//     PlcTask Outputs/G_IO.arDO[20]/Ch[11] <-> DO0/0016ETP Output-bit maping/Digital output CH2-bit3
//     PlcTask Outputs/G_IO.arDO[20]/Ch[12] <-> DO0/0016ETP Output-bit maping/Digital output CH2-bit4
//     PlcTask Outputs/G_IO.arDO[20]/Ch[13] <-> DO0/0016ETP Output-bit maping/Digital output CH2-bit5
//     PlcTask Outputs/G_IO.arDO[20]/Ch[14] <-> DO0/0016ETP Output-bit maping/Digital output CH2-bit6
//     PlcTask Outputs/G_IO.arDO[20]/Ch[15] <-> DO0/0016ETP Output-bit maping/Digital output CH2-bit7
//     PlcTask Outputs/G_IO.arDO[20]/Ch[1] <-> DO0/0016ETP Output-bit maping/Digital output CH1-bit1
//     PlcTask Outputs/G_IO.arDO[20]/Ch[2] <-> DO0/0016ETP Output-bit maping/Digital output CH1-bit2
//     PlcTask Outputs/G_IO.arDO[20]/Ch[3] <-> DO0/0016ETP Output-bit maping/Digital output CH1-bit3
//     PlcTask Outputs/G_IO.arDO[20]/Ch[4] <-> DO0/0016ETP Output-bit maping/Digital output CH1-bit4
//     PlcTask Outputs/G_IO.arDO[20]/Ch[5] <-> DO0/0016ETP Output-bit maping/Digital output CH1-bit5
//     PlcTask Outputs/G_IO.arDO[20]/Ch[6] <-> DO0/0016ETP Output-bit maping/Digital output CH1-bit6
//     PlcTask Outputs/G_IO.arDO[20]/Ch[7] <-> DO0/0016ETP Output-bit maping/Digital output CH1-bit7
//     PlcTask Outputs/G_IO.arDO[20]/Ch[8] <-> DO0/0016ETP Output-bit maping/Digital output CH2-bit0
//     PlcTask Outputs/G_IO.arDO[20]/Ch[9] <-> DO0/0016ETP Output-bit maping/Digital output CH2-bit1
//     PlcTask Outputs/G_IO.arDO[21]/Ch[0] <-> DO1/0016ETP Output-bit maping/Digital output CH1-bit0
//     PlcTask Outputs/G_IO.arDO[21]/Ch[10] <-> DO1/0016ETP Output-bit maping/Digital output CH2-bit2
//     PlcTask Outputs/G_IO.arDO[21]/Ch[11] <-> DO1/0016ETP Output-bit maping/Digital output CH2-bit3
//     PlcTask Outputs/G_IO.arDO[21]/Ch[12] <-> DO1/0016ETP Output-bit maping/Digital output CH2-bit4
//     PlcTask Outputs/G_IO.arDO[21]/Ch[13] <-> DO1/0016ETP Output-bit maping/Digital output CH2-bit5
//     PlcTask Outputs/G_IO.arDO[21]/Ch[14] <-> DO1/0016ETP Output-bit maping/Digital output CH2-bit6
//     PlcTask Outputs/G_IO.arDO[21]/Ch[15] <-> DO1/0016ETP Output-bit maping/Digital output CH2-bit7
//     PlcTask Outputs/G_IO.arDO[21]/Ch[1] <-> DO1/0016ETP Output-bit maping/Digital output CH1-bit1
//     PlcTask Outputs/G_IO.arDO[21]/Ch[2] <-> DO1/0016ETP Output-bit maping/Digital output CH1-bit2
//     PlcTask Outputs/G_IO.arDO[21]/Ch[3] <-> DO1/0016ETP Output-bit maping/Digital output CH1-bit3
//     PlcTask Outputs/G_IO.arDO[21]/Ch[4] <-> DO1/0016ETP Output-bit maping/Digital output CH1-bit4
//     PlcTask Outputs/G_IO.arDO[21]/Ch[5] <-> DO1/0016ETP Output-bit maping/Digital output CH1-bit5
//     PlcTask Outputs/G_IO.arDO[21]/Ch[6] <-> DO1/0016ETP Output-bit maping/Digital output CH1-bit6
//     PlcTask Outputs/G_IO.arDO[21]/Ch[7] <-> DO1/0016ETP Output-bit maping/Digital output CH1-bit7
//     PlcTask Outputs/G_IO.arDO[21]/Ch[8] <-> DO1/0016ETP Output-bit maping/Digital output CH2-bit0
//     PlcTask Outputs/G_IO.arDO[21]/Ch[9] <-> DO1/0016ETP Output-bit maping/Digital output CH2-bit1
//   kittingDeca/kittingDeca Instance <-> rem_wf/rem5_valve
//     PlcTask Outputs/G_IO.arDO[22]/Ch[0] <-> Module 1 (C2S-EC-24B)/Outputs/valve[1..4][0]
//     PlcTask Outputs/G_IO.arDO[22]/Ch[10] <-> Module 1 (C2S-EC-24B)/Outputs/valve[5..8][2]
//     PlcTask Outputs/G_IO.arDO[22]/Ch[11] <-> Module 1 (C2S-EC-24B)/Outputs/valve[5..8][3]
//     PlcTask Outputs/G_IO.arDO[22]/Ch[12] <-> Module 1 (C2S-EC-24B)/Outputs/valve[5..8][4]
//     PlcTask Outputs/G_IO.arDO[22]/Ch[13] <-> Module 1 (C2S-EC-24B)/Outputs/valve[5..8][5]
//     PlcTask Outputs/G_IO.arDO[22]/Ch[14] <-> Module 1 (C2S-EC-24B)/Outputs/valve[5..8][6]
//     PlcTask Outputs/G_IO.arDO[22]/Ch[15] <-> Module 1 (C2S-EC-24B)/Outputs/valve[5..8][7]
//     PlcTask Outputs/G_IO.arDO[22]/Ch[1] <-> Module 1 (C2S-EC-24B)/Outputs/valve[1..4][1]
//     PlcTask Outputs/G_IO.arDO[22]/Ch[2] <-> Module 1 (C2S-EC-24B)/Outputs/valve[1..4][2]
//     PlcTask Outputs/G_IO.arDO[22]/Ch[3] <-> Module 1 (C2S-EC-24B)/Outputs/valve[1..4][3]
//     PlcTask Outputs/G_IO.arDO[22]/Ch[4] <-> Module 1 (C2S-EC-24B)/Outputs/valve[1..4][4]
//     PlcTask Outputs/G_IO.arDO[22]/Ch[5] <-> Module 1 (C2S-EC-24B)/Outputs/valve[1..4][5]
//     PlcTask Outputs/G_IO.arDO[22]/Ch[6] <-> Module 1 (C2S-EC-24B)/Outputs/valve[1..4][6]
//     PlcTask Outputs/G_IO.arDO[22]/Ch[7] <-> Module 1 (C2S-EC-24B)/Outputs/valve[1..4][7]
//     PlcTask Outputs/G_IO.arDO[22]/Ch[8] <-> Module 1 (C2S-EC-24B)/Outputs/valve[5..8][0]
//     PlcTask Outputs/G_IO.arDO[22]/Ch[9] <-> Module 1 (C2S-EC-24B)/Outputs/valve[5..8][1]
//     PlcTask Outputs/G_IO.arDO[23]/Ch[0] <-> Module 1 (C2S-EC-24B)/Outputs/valve[9..12][0]
//     PlcTask Outputs/G_IO.arDO[23]/Ch[1] <-> Module 1 (C2S-EC-24B)/Outputs/valve[9..12][1]
//     PlcTask Outputs/G_IO.arDO[23]/Ch[2] <-> Module 1 (C2S-EC-24B)/Outputs/valve[9..12][2]
//     PlcTask Outputs/G_IO.arDO[23]/Ch[3] <-> Module 1 (C2S-EC-24B)/Outputs/valve[9..12][3]
//     PlcTask Outputs/G_IO.arDO[23]/Ch[4] <-> Module 1 (C2S-EC-24B)/Outputs/valve[9..12][4]
//     PlcTask Outputs/G_IO.arDO[23]/Ch[5] <-> Module 1 (C2S-EC-24B)/Outputs/valve[9..12][5]
//     PlcTask Outputs/G_IO.arDO[23]/Ch[6] <-> Module 1 (C2S-EC-24B)/Outputs/valve[9..12][6]
//     PlcTask Outputs/G_IO.arDO[23]/Ch[7] <-> Module 1 (C2S-EC-24B)/Outputs/valve[9..12][7]
//   kittingDeca/kittingDeca Instance <-> rem_wf/rem6_dio
//     PlcTask Inputs/G_IO.arDI[24]/Ch[0] <-> DI0/1600END input-bit maping/Digital input CH1-bit0
//     PlcTask Inputs/G_IO.arDI[24]/Ch[10] <-> DI0/1600END input-bit maping/Digital input CH2-bit2
//     PlcTask Inputs/G_IO.arDI[24]/Ch[11] <-> DI0/1600END input-bit maping/Digital input CH2-bit3
//     PlcTask Inputs/G_IO.arDI[24]/Ch[12] <-> DI0/1600END input-bit maping/Digital input CH2-bit4
//     PlcTask Inputs/G_IO.arDI[24]/Ch[13] <-> DI0/1600END input-bit maping/Digital input CH2-bit5
//     PlcTask Inputs/G_IO.arDI[24]/Ch[14] <-> DI0/1600END input-bit maping/Digital input CH2-bit6
//     PlcTask Inputs/G_IO.arDI[24]/Ch[15] <-> DI0/1600END input-bit maping/Digital input CH2-bit7
//     PlcTask Inputs/G_IO.arDI[24]/Ch[1] <-> DI0/1600END input-bit maping/Digital input CH1-bit1
//     PlcTask Inputs/G_IO.arDI[24]/Ch[2] <-> DI0/1600END input-bit maping/Digital input CH1-bit2
//     PlcTask Inputs/G_IO.arDI[24]/Ch[3] <-> DI0/1600END input-bit maping/Digital input CH1-bit3
//     PlcTask Inputs/G_IO.arDI[24]/Ch[4] <-> DI0/1600END input-bit maping/Digital input CH1-bit4
//     PlcTask Inputs/G_IO.arDI[24]/Ch[5] <-> DI0/1600END input-bit maping/Digital input CH1-bit5
//     PlcTask Inputs/G_IO.arDI[24]/Ch[6] <-> DI0/1600END input-bit maping/Digital input CH1-bit6
//     PlcTask Inputs/G_IO.arDI[24]/Ch[7] <-> DI0/1600END input-bit maping/Digital input CH1-bit7
//     PlcTask Inputs/G_IO.arDI[24]/Ch[8] <-> DI0/1600END input-bit maping/Digital input CH2-bit0
//     PlcTask Inputs/G_IO.arDI[24]/Ch[9] <-> DI0/1600END input-bit maping/Digital input CH2-bit1
//     PlcTask Inputs/G_IO.arDI[25]/Ch[0] <-> DI1/1600END input-bit maping/Digital input CH1-bit0
//     PlcTask Inputs/G_IO.arDI[25]/Ch[10] <-> DI1/1600END input-bit maping/Digital input CH2-bit2
//     PlcTask Inputs/G_IO.arDI[25]/Ch[11] <-> DI1/1600END input-bit maping/Digital input CH2-bit3
//     PlcTask Inputs/G_IO.arDI[25]/Ch[12] <-> DI1/1600END input-bit maping/Digital input CH2-bit4
//     PlcTask Inputs/G_IO.arDI[25]/Ch[13] <-> DI1/1600END input-bit maping/Digital input CH2-bit5
//     PlcTask Inputs/G_IO.arDI[25]/Ch[14] <-> DI1/1600END input-bit maping/Digital input CH2-bit6
//     PlcTask Inputs/G_IO.arDI[25]/Ch[15] <-> DI1/1600END input-bit maping/Digital input CH2-bit7
//     PlcTask Inputs/G_IO.arDI[25]/Ch[1] <-> DI1/1600END input-bit maping/Digital input CH1-bit1
//     PlcTask Inputs/G_IO.arDI[25]/Ch[2] <-> DI1/1600END input-bit maping/Digital input CH1-bit2
//     PlcTask Inputs/G_IO.arDI[25]/Ch[3] <-> DI1/1600END input-bit maping/Digital input CH1-bit3
//     PlcTask Inputs/G_IO.arDI[25]/Ch[4] <-> DI1/1600END input-bit maping/Digital input CH1-bit4
//     PlcTask Inputs/G_IO.arDI[25]/Ch[5] <-> DI1/1600END input-bit maping/Digital input CH1-bit5
//     PlcTask Inputs/G_IO.arDI[25]/Ch[6] <-> DI1/1600END input-bit maping/Digital input CH1-bit6
//     PlcTask Inputs/G_IO.arDI[25]/Ch[7] <-> DI1/1600END input-bit maping/Digital input CH1-bit7
//     PlcTask Inputs/G_IO.arDI[25]/Ch[8] <-> DI1/1600END input-bit maping/Digital input CH2-bit0
//     PlcTask Inputs/G_IO.arDI[25]/Ch[9] <-> DI1/1600END input-bit maping/Digital input CH2-bit1
//     PlcTask Inputs/G_IO.arDI[26]/Ch[0] <-> DI2/1600END input-bit maping/Digital input CH1-bit0
//     PlcTask Inputs/G_IO.arDI[26]/Ch[10] <-> DI2/1600END input-bit maping/Digital input CH2-bit2
//     PlcTask Inputs/G_IO.arDI[26]/Ch[11] <-> DI2/1600END input-bit maping/Digital input CH2-bit3
//     PlcTask Inputs/G_IO.arDI[26]/Ch[12] <-> DI2/1600END input-bit maping/Digital input CH2-bit4
//     PlcTask Inputs/G_IO.arDI[26]/Ch[13] <-> DI2/1600END input-bit maping/Digital input CH2-bit5
//     PlcTask Inputs/G_IO.arDI[26]/Ch[14] <-> DI2/1600END input-bit maping/Digital input CH2-bit6
//     PlcTask Inputs/G_IO.arDI[26]/Ch[15] <-> DI2/1600END input-bit maping/Digital input CH2-bit7
//     PlcTask Inputs/G_IO.arDI[26]/Ch[1] <-> DI2/1600END input-bit maping/Digital input CH1-bit1
//     PlcTask Inputs/G_IO.arDI[26]/Ch[2] <-> DI2/1600END input-bit maping/Digital input CH1-bit2
//     PlcTask Inputs/G_IO.arDI[26]/Ch[3] <-> DI2/1600END input-bit maping/Digital input CH1-bit3
//     PlcTask Inputs/G_IO.arDI[26]/Ch[4] <-> DI2/1600END input-bit maping/Digital input CH1-bit4
//     PlcTask Inputs/G_IO.arDI[26]/Ch[5] <-> DI2/1600END input-bit maping/Digital input CH1-bit5
//     PlcTask Inputs/G_IO.arDI[26]/Ch[6] <-> DI2/1600END input-bit maping/Digital input CH1-bit6
//     PlcTask Inputs/G_IO.arDI[26]/Ch[7] <-> DI2/1600END input-bit maping/Digital input CH1-bit7
//     PlcTask Inputs/G_IO.arDI[26]/Ch[8] <-> DI2/1600END input-bit maping/Digital input CH2-bit0
//     PlcTask Inputs/G_IO.arDI[26]/Ch[9] <-> DI2/1600END input-bit maping/Digital input CH2-bit1
//     PlcTask Inputs/G_IO.arDI[27]/Ch[0] <-> DI3/1600END input-bit maping/Digital input CH1-bit0
//     PlcTask Inputs/G_IO.arDI[27]/Ch[10] <-> DI3/1600END input-bit maping/Digital input CH2-bit2
//     PlcTask Inputs/G_IO.arDI[27]/Ch[11] <-> DI3/1600END input-bit maping/Digital input CH2-bit3
//     PlcTask Inputs/G_IO.arDI[27]/Ch[12] <-> DI3/1600END input-bit maping/Digital input CH2-bit4
//     PlcTask Inputs/G_IO.arDI[27]/Ch[13] <-> DI3/1600END input-bit maping/Digital input CH2-bit5
//     PlcTask Inputs/G_IO.arDI[27]/Ch[14] <-> DI3/1600END input-bit maping/Digital input CH2-bit6
//     PlcTask Inputs/G_IO.arDI[27]/Ch[15] <-> DI3/1600END input-bit maping/Digital input CH2-bit7
//     PlcTask Inputs/G_IO.arDI[27]/Ch[1] <-> DI3/1600END input-bit maping/Digital input CH1-bit1
//     PlcTask Inputs/G_IO.arDI[27]/Ch[2] <-> DI3/1600END input-bit maping/Digital input CH1-bit2
//     PlcTask Inputs/G_IO.arDI[27]/Ch[3] <-> DI3/1600END input-bit maping/Digital input CH1-bit3
//     PlcTask Inputs/G_IO.arDI[27]/Ch[4] <-> DI3/1600END input-bit maping/Digital input CH1-bit4
//     PlcTask Inputs/G_IO.arDI[27]/Ch[5] <-> DI3/1600END input-bit maping/Digital input CH1-bit5
//     PlcTask Inputs/G_IO.arDI[27]/Ch[6] <-> DI3/1600END input-bit maping/Digital input CH1-bit6
//     PlcTask Inputs/G_IO.arDI[27]/Ch[7] <-> DI3/1600END input-bit maping/Digital input CH1-bit7
//     PlcTask Inputs/G_IO.arDI[27]/Ch[8] <-> DI3/1600END input-bit maping/Digital input CH2-bit0
//     PlcTask Inputs/G_IO.arDI[27]/Ch[9] <-> DI3/1600END input-bit maping/Digital input CH2-bit1
//     PlcTask Outputs/G_IO.arDO[24]/Ch[0] <-> DO0/0016ETP Output-bit maping/Digital output CH1-bit0
//     PlcTask Outputs/G_IO.arDO[24]/Ch[10] <-> DO0/0016ETP Output-bit maping/Digital output CH2-bit2
//     PlcTask Outputs/G_IO.arDO[24]/Ch[11] <-> DO0/0016ETP Output-bit maping/Digital output CH2-bit3
//     PlcTask Outputs/G_IO.arDO[24]/Ch[12] <-> DO0/0016ETP Output-bit maping/Digital output CH2-bit4
//     PlcTask Outputs/G_IO.arDO[24]/Ch[13] <-> DO0/0016ETP Output-bit maping/Digital output CH2-bit5
//     PlcTask Outputs/G_IO.arDO[24]/Ch[14] <-> DO0/0016ETP Output-bit maping/Digital output CH2-bit6
//     PlcTask Outputs/G_IO.arDO[24]/Ch[15] <-> DO0/0016ETP Output-bit maping/Digital output CH2-bit7
//     PlcTask Outputs/G_IO.arDO[24]/Ch[1] <-> DO0/0016ETP Output-bit maping/Digital output CH1-bit1
//     PlcTask Outputs/G_IO.arDO[24]/Ch[2] <-> DO0/0016ETP Output-bit maping/Digital output CH1-bit2
//     PlcTask Outputs/G_IO.arDO[24]/Ch[3] <-> DO0/0016ETP Output-bit maping/Digital output CH1-bit3
//     PlcTask Outputs/G_IO.arDO[24]/Ch[4] <-> DO0/0016ETP Output-bit maping/Digital output CH1-bit4
//     PlcTask Outputs/G_IO.arDO[24]/Ch[5] <-> DO0/0016ETP Output-bit maping/Digital output CH1-bit5
//     PlcTask Outputs/G_IO.arDO[24]/Ch[6] <-> DO0/0016ETP Output-bit maping/Digital output CH1-bit6
//     PlcTask Outputs/G_IO.arDO[24]/Ch[7] <-> DO0/0016ETP Output-bit maping/Digital output CH1-bit7
//     PlcTask Outputs/G_IO.arDO[24]/Ch[8] <-> DO0/0016ETP Output-bit maping/Digital output CH2-bit0
//     PlcTask Outputs/G_IO.arDO[24]/Ch[9] <-> DO0/0016ETP Output-bit maping/Digital output CH2-bit1
//     PlcTask Outputs/G_IO.arDO[25]/Ch[0] <-> DO1/0016ETP Output-bit maping/Digital output CH1-bit0
//     PlcTask Outputs/G_IO.arDO[25]/Ch[10] <-> DO1/0016ETP Output-bit maping/Digital output CH2-bit2
//     PlcTask Outputs/G_IO.arDO[25]/Ch[11] <-> DO1/0016ETP Output-bit maping/Digital output CH2-bit3
//     PlcTask Outputs/G_IO.arDO[25]/Ch[12] <-> DO1/0016ETP Output-bit maping/Digital output CH2-bit4
//     PlcTask Outputs/G_IO.arDO[25]/Ch[13] <-> DO1/0016ETP Output-bit maping/Digital output CH2-bit5
//     PlcTask Outputs/G_IO.arDO[25]/Ch[14] <-> DO1/0016ETP Output-bit maping/Digital output CH2-bit6
//     PlcTask Outputs/G_IO.arDO[25]/Ch[15] <-> DO1/0016ETP Output-bit maping/Digital output CH2-bit7
//     PlcTask Outputs/G_IO.arDO[25]/Ch[1] <-> DO1/0016ETP Output-bit maping/Digital output CH1-bit1
//     PlcTask Outputs/G_IO.arDO[25]/Ch[2] <-> DO1/0016ETP Output-bit maping/Digital output CH1-bit2
//     PlcTask Outputs/G_IO.arDO[25]/Ch[3] <-> DO1/0016ETP Output-bit maping/Digital output CH1-bit3
//     PlcTask Outputs/G_IO.arDO[25]/Ch[4] <-> DO1/0016ETP Output-bit maping/Digital output CH1-bit4
//     PlcTask Outputs/G_IO.arDO[25]/Ch[5] <-> DO1/0016ETP Output-bit maping/Digital output CH1-bit5
//     PlcTask Outputs/G_IO.arDO[25]/Ch[6] <-> DO1/0016ETP Output-bit maping/Digital output CH1-bit6
//     PlcTask Outputs/G_IO.arDO[25]/Ch[7] <-> DO1/0016ETP Output-bit maping/Digital output CH1-bit7
//     PlcTask Outputs/G_IO.arDO[25]/Ch[8] <-> DO1/0016ETP Output-bit maping/Digital output CH2-bit0
//     PlcTask Outputs/G_IO.arDO[25]/Ch[9] <-> DO1/0016ETP Output-bit maping/Digital output CH2-bit1
//   kittingDeca/kittingDeca Instance <-> rem_wf/rem6_valve
//     PlcTask Outputs/G_IO.arDO[26]/Ch[0] <-> Module 1 (C2S-EC-24B)/Outputs/valve[1..4][0]
//     PlcTask Outputs/G_IO.arDO[26]/Ch[10] <-> Module 1 (C2S-EC-24B)/Outputs/valve[5..8][2]
//     PlcTask Outputs/G_IO.arDO[26]/Ch[11] <-> Module 1 (C2S-EC-24B)/Outputs/valve[5..8][3]
//     PlcTask Outputs/G_IO.arDO[26]/Ch[12] <-> Module 1 (C2S-EC-24B)/Outputs/valve[5..8][4]
//     PlcTask Outputs/G_IO.arDO[26]/Ch[13] <-> Module 1 (C2S-EC-24B)/Outputs/valve[5..8][5]
//     PlcTask Outputs/G_IO.arDO[26]/Ch[14] <-> Module 1 (C2S-EC-24B)/Outputs/valve[5..8][6]
//     PlcTask Outputs/G_IO.arDO[26]/Ch[15] <-> Module 1 (C2S-EC-24B)/Outputs/valve[5..8][7]
//     PlcTask Outputs/G_IO.arDO[26]/Ch[1] <-> Module 1 (C2S-EC-24B)/Outputs/valve[1..4][1]
//     PlcTask Outputs/G_IO.arDO[26]/Ch[2] <-> Module 1 (C2S-EC-24B)/Outputs/valve[1..4][2]
//     PlcTask Outputs/G_IO.arDO[26]/Ch[3] <-> Module 1 (C2S-EC-24B)/Outputs/valve[1..4][3]
//     PlcTask Outputs/G_IO.arDO[26]/Ch[4] <-> Module 1 (C2S-EC-24B)/Outputs/valve[1..4][4]
//     PlcTask Outputs/G_IO.arDO[26]/Ch[5] <-> Module 1 (C2S-EC-24B)/Outputs/valve[1..4][5]
//     PlcTask Outputs/G_IO.arDO[26]/Ch[6] <-> Module 1 (C2S-EC-24B)/Outputs/valve[1..4][6]
//     PlcTask Outputs/G_IO.arDO[26]/Ch[7] <-> Module 1 (C2S-EC-24B)/Outputs/valve[1..4][7]
//     PlcTask Outputs/G_IO.arDO[26]/Ch[8] <-> Module 1 (C2S-EC-24B)/Outputs/valve[5..8][0]
//     PlcTask Outputs/G_IO.arDO[26]/Ch[9] <-> Module 1 (C2S-EC-24B)/Outputs/valve[5..8][1]
//     PlcTask Outputs/G_IO.arDO[27]/Ch[0] <-> Module 1 (C2S-EC-24B)/Outputs/valve[9..12][0]
//     PlcTask Outputs/G_IO.arDO[27]/Ch[1] <-> Module 1 (C2S-EC-24B)/Outputs/valve[9..12][1]
//     PlcTask Outputs/G_IO.arDO[27]/Ch[2] <-> Module 1 (C2S-EC-24B)/Outputs/valve[9..12][2]
//     PlcTask Outputs/G_IO.arDO[27]/Ch[3] <-> Module 1 (C2S-EC-24B)/Outputs/valve[9..12][3]
//     PlcTask Outputs/G_IO.arDO[27]/Ch[4] <-> Module 1 (C2S-EC-24B)/Outputs/valve[9..12][4]
//     PlcTask Outputs/G_IO.arDO[27]/Ch[5] <-> Module 1 (C2S-EC-24B)/Outputs/valve[9..12][5]
//     PlcTask Outputs/G_IO.arDO[27]/Ch[6] <-> Module 1 (C2S-EC-24B)/Outputs/valve[9..12][6]
//     PlcTask Outputs/G_IO.arDO[27]/Ch[7] <-> Module 1 (C2S-EC-24B)/Outputs/valve[9..12][7]
//   kittingDeca/kittingDeca Instance <-> rem_wf/rem7_dio
//     PlcTask Inputs/G_IO.arDI[28]/Ch[0] <-> DI0/1600END input-bit maping/Digital input CH1-bit0
//     PlcTask Inputs/G_IO.arDI[28]/Ch[10] <-> DI0/1600END input-bit maping/Digital input CH2-bit2
//     PlcTask Inputs/G_IO.arDI[28]/Ch[11] <-> DI0/1600END input-bit maping/Digital input CH2-bit3
//     PlcTask Inputs/G_IO.arDI[28]/Ch[12] <-> DI0/1600END input-bit maping/Digital input CH2-bit4
//     PlcTask Inputs/G_IO.arDI[28]/Ch[13] <-> DI0/1600END input-bit maping/Digital input CH2-bit5
//     PlcTask Inputs/G_IO.arDI[28]/Ch[14] <-> DI0/1600END input-bit maping/Digital input CH2-bit6
//     PlcTask Inputs/G_IO.arDI[28]/Ch[15] <-> DI0/1600END input-bit maping/Digital input CH2-bit7
//     PlcTask Inputs/G_IO.arDI[28]/Ch[1] <-> DI0/1600END input-bit maping/Digital input CH1-bit1
//     PlcTask Inputs/G_IO.arDI[28]/Ch[2] <-> DI0/1600END input-bit maping/Digital input CH1-bit2
//     PlcTask Inputs/G_IO.arDI[28]/Ch[3] <-> DI0/1600END input-bit maping/Digital input CH1-bit3
//     PlcTask Inputs/G_IO.arDI[28]/Ch[4] <-> DI0/1600END input-bit maping/Digital input CH1-bit4
//     PlcTask Inputs/G_IO.arDI[28]/Ch[5] <-> DI0/1600END input-bit maping/Digital input CH1-bit5
//     PlcTask Inputs/G_IO.arDI[28]/Ch[6] <-> DI0/1600END input-bit maping/Digital input CH1-bit6
//     PlcTask Inputs/G_IO.arDI[28]/Ch[7] <-> DI0/1600END input-bit maping/Digital input CH1-bit7
//     PlcTask Inputs/G_IO.arDI[28]/Ch[8] <-> DI0/1600END input-bit maping/Digital input CH2-bit0
//     PlcTask Inputs/G_IO.arDI[28]/Ch[9] <-> DI0/1600END input-bit maping/Digital input CH2-bit1
//     PlcTask Inputs/G_IO.arDI[29]/Ch[0] <-> DI1/1600END input-bit maping/Digital input CH1-bit0
//     PlcTask Inputs/G_IO.arDI[29]/Ch[10] <-> DI1/1600END input-bit maping/Digital input CH2-bit2
//     PlcTask Inputs/G_IO.arDI[29]/Ch[11] <-> DI1/1600END input-bit maping/Digital input CH2-bit3
//     PlcTask Inputs/G_IO.arDI[29]/Ch[12] <-> DI1/1600END input-bit maping/Digital input CH2-bit4
//     PlcTask Inputs/G_IO.arDI[29]/Ch[13] <-> DI1/1600END input-bit maping/Digital input CH2-bit5
//     PlcTask Inputs/G_IO.arDI[29]/Ch[14] <-> DI1/1600END input-bit maping/Digital input CH2-bit6
//     PlcTask Inputs/G_IO.arDI[29]/Ch[15] <-> DI1/1600END input-bit maping/Digital input CH2-bit7
//     PlcTask Inputs/G_IO.arDI[29]/Ch[1] <-> DI1/1600END input-bit maping/Digital input CH1-bit1
//     PlcTask Inputs/G_IO.arDI[29]/Ch[2] <-> DI1/1600END input-bit maping/Digital input CH1-bit2
//     PlcTask Inputs/G_IO.arDI[29]/Ch[3] <-> DI1/1600END input-bit maping/Digital input CH1-bit3
//     PlcTask Inputs/G_IO.arDI[29]/Ch[4] <-> DI1/1600END input-bit maping/Digital input CH1-bit4
//     PlcTask Inputs/G_IO.arDI[29]/Ch[5] <-> DI1/1600END input-bit maping/Digital input CH1-bit5
//     PlcTask Inputs/G_IO.arDI[29]/Ch[6] <-> DI1/1600END input-bit maping/Digital input CH1-bit6
//     PlcTask Inputs/G_IO.arDI[29]/Ch[7] <-> DI1/1600END input-bit maping/Digital input CH1-bit7
//     PlcTask Inputs/G_IO.arDI[29]/Ch[8] <-> DI1/1600END input-bit maping/Digital input CH2-bit0
//     PlcTask Inputs/G_IO.arDI[29]/Ch[9] <-> DI1/1600END input-bit maping/Digital input CH2-bit1
//     PlcTask Inputs/G_IO.arDI[30]/Ch[0] <-> DI2/1600END input-bit maping/Digital input CH1-bit0
//     PlcTask Inputs/G_IO.arDI[30]/Ch[10] <-> DI2/1600END input-bit maping/Digital input CH2-bit2
//     PlcTask Inputs/G_IO.arDI[30]/Ch[11] <-> DI2/1600END input-bit maping/Digital input CH2-bit3
//     PlcTask Inputs/G_IO.arDI[30]/Ch[12] <-> DI2/1600END input-bit maping/Digital input CH2-bit4
//     PlcTask Inputs/G_IO.arDI[30]/Ch[13] <-> DI2/1600END input-bit maping/Digital input CH2-bit5
//     PlcTask Inputs/G_IO.arDI[30]/Ch[14] <-> DI2/1600END input-bit maping/Digital input CH2-bit6
//     PlcTask Inputs/G_IO.arDI[30]/Ch[15] <-> DI2/1600END input-bit maping/Digital input CH2-bit7
//     PlcTask Inputs/G_IO.arDI[30]/Ch[1] <-> DI2/1600END input-bit maping/Digital input CH1-bit1
//     PlcTask Inputs/G_IO.arDI[30]/Ch[2] <-> DI2/1600END input-bit maping/Digital input CH1-bit2
//     PlcTask Inputs/G_IO.arDI[30]/Ch[3] <-> DI2/1600END input-bit maping/Digital input CH1-bit3
//     PlcTask Inputs/G_IO.arDI[30]/Ch[4] <-> DI2/1600END input-bit maping/Digital input CH1-bit4
//     PlcTask Inputs/G_IO.arDI[30]/Ch[5] <-> DI2/1600END input-bit maping/Digital input CH1-bit5
//     PlcTask Inputs/G_IO.arDI[30]/Ch[6] <-> DI2/1600END input-bit maping/Digital input CH1-bit6
//     PlcTask Inputs/G_IO.arDI[30]/Ch[7] <-> DI2/1600END input-bit maping/Digital input CH1-bit7
//     PlcTask Inputs/G_IO.arDI[30]/Ch[8] <-> DI2/1600END input-bit maping/Digital input CH2-bit0
//     PlcTask Inputs/G_IO.arDI[30]/Ch[9] <-> DI2/1600END input-bit maping/Digital input CH2-bit1
//     PlcTask Inputs/G_IO.arDI[31]/Ch[0] <-> DI3/1600END input-bit maping/Digital input CH1-bit0
//     PlcTask Inputs/G_IO.arDI[31]/Ch[10] <-> DI3/1600END input-bit maping/Digital input CH2-bit2
//     PlcTask Inputs/G_IO.arDI[31]/Ch[11] <-> DI3/1600END input-bit maping/Digital input CH2-bit3
//     PlcTask Inputs/G_IO.arDI[31]/Ch[12] <-> DI3/1600END input-bit maping/Digital input CH2-bit4
//     PlcTask Inputs/G_IO.arDI[31]/Ch[13] <-> DI3/1600END input-bit maping/Digital input CH2-bit5
//     PlcTask Inputs/G_IO.arDI[31]/Ch[14] <-> DI3/1600END input-bit maping/Digital input CH2-bit6
//     PlcTask Inputs/G_IO.arDI[31]/Ch[15] <-> DI3/1600END input-bit maping/Digital input CH2-bit7
//     PlcTask Inputs/G_IO.arDI[31]/Ch[1] <-> DI3/1600END input-bit maping/Digital input CH1-bit1
//     PlcTask Inputs/G_IO.arDI[31]/Ch[2] <-> DI3/1600END input-bit maping/Digital input CH1-bit2
//     PlcTask Inputs/G_IO.arDI[31]/Ch[3] <-> DI3/1600END input-bit maping/Digital input CH1-bit3
//     PlcTask Inputs/G_IO.arDI[31]/Ch[4] <-> DI3/1600END input-bit maping/Digital input CH1-bit4
//     PlcTask Inputs/G_IO.arDI[31]/Ch[5] <-> DI3/1600END input-bit maping/Digital input CH1-bit5
//     PlcTask Inputs/G_IO.arDI[31]/Ch[6] <-> DI3/1600END input-bit maping/Digital input CH1-bit6
//     PlcTask Inputs/G_IO.arDI[31]/Ch[7] <-> DI3/1600END input-bit maping/Digital input CH1-bit7
//     PlcTask Inputs/G_IO.arDI[31]/Ch[8] <-> DI3/1600END input-bit maping/Digital input CH2-bit0
//     PlcTask Inputs/G_IO.arDI[31]/Ch[9] <-> DI3/1600END input-bit maping/Digital input CH2-bit1
//     PlcTask Outputs/G_IO.arDO[28]/Ch[0] <-> DO0/0016ETP Output-bit maping/Digital output CH1-bit0
//     PlcTask Outputs/G_IO.arDO[28]/Ch[10] <-> DO0/0016ETP Output-bit maping/Digital output CH2-bit2
//     PlcTask Outputs/G_IO.arDO[28]/Ch[11] <-> DO0/0016ETP Output-bit maping/Digital output CH2-bit3
//     PlcTask Outputs/G_IO.arDO[28]/Ch[12] <-> DO0/0016ETP Output-bit maping/Digital output CH2-bit4
//     PlcTask Outputs/G_IO.arDO[28]/Ch[13] <-> DO0/0016ETP Output-bit maping/Digital output CH2-bit5
//     PlcTask Outputs/G_IO.arDO[28]/Ch[14] <-> DO0/0016ETP Output-bit maping/Digital output CH2-bit6
//     PlcTask Outputs/G_IO.arDO[28]/Ch[15] <-> DO0/0016ETP Output-bit maping/Digital output CH2-bit7
//     PlcTask Outputs/G_IO.arDO[28]/Ch[1] <-> DO0/0016ETP Output-bit maping/Digital output CH1-bit1
//     PlcTask Outputs/G_IO.arDO[28]/Ch[2] <-> DO0/0016ETP Output-bit maping/Digital output CH1-bit2
//     PlcTask Outputs/G_IO.arDO[28]/Ch[3] <-> DO0/0016ETP Output-bit maping/Digital output CH1-bit3
//     PlcTask Outputs/G_IO.arDO[28]/Ch[4] <-> DO0/0016ETP Output-bit maping/Digital output CH1-bit4
//     PlcTask Outputs/G_IO.arDO[28]/Ch[5] <-> DO0/0016ETP Output-bit maping/Digital output CH1-bit5
//     PlcTask Outputs/G_IO.arDO[28]/Ch[6] <-> DO0/0016ETP Output-bit maping/Digital output CH1-bit6
//     PlcTask Outputs/G_IO.arDO[28]/Ch[7] <-> DO0/0016ETP Output-bit maping/Digital output CH1-bit7
//     PlcTask Outputs/G_IO.arDO[28]/Ch[8] <-> DO0/0016ETP Output-bit maping/Digital output CH2-bit0
//     PlcTask Outputs/G_IO.arDO[28]/Ch[9] <-> DO0/0016ETP Output-bit maping/Digital output CH2-bit1
//     PlcTask Outputs/G_IO.arDO[29]/Ch[0] <-> DO1/0016ETP Output-bit maping/Digital output CH1-bit0
//     PlcTask Outputs/G_IO.arDO[29]/Ch[10] <-> DO1/0016ETP Output-bit maping/Digital output CH2-bit2
//     PlcTask Outputs/G_IO.arDO[29]/Ch[11] <-> DO1/0016ETP Output-bit maping/Digital output CH2-bit3
//     PlcTask Outputs/G_IO.arDO[29]/Ch[12] <-> DO1/0016ETP Output-bit maping/Digital output CH2-bit4
//     PlcTask Outputs/G_IO.arDO[29]/Ch[13] <-> DO1/0016ETP Output-bit maping/Digital output CH2-bit5
//     PlcTask Outputs/G_IO.arDO[29]/Ch[14] <-> DO1/0016ETP Output-bit maping/Digital output CH2-bit6
//     PlcTask Outputs/G_IO.arDO[29]/Ch[15] <-> DO1/0016ETP Output-bit maping/Digital output CH2-bit7
//     PlcTask Outputs/G_IO.arDO[29]/Ch[1] <-> DO1/0016ETP Output-bit maping/Digital output CH1-bit1
//     PlcTask Outputs/G_IO.arDO[29]/Ch[2] <-> DO1/0016ETP Output-bit maping/Digital output CH1-bit2
//     PlcTask Outputs/G_IO.arDO[29]/Ch[3] <-> DO1/0016ETP Output-bit maping/Digital output CH1-bit3
//     PlcTask Outputs/G_IO.arDO[29]/Ch[4] <-> DO1/0016ETP Output-bit maping/Digital output CH1-bit4
//     PlcTask Outputs/G_IO.arDO[29]/Ch[5] <-> DO1/0016ETP Output-bit maping/Digital output CH1-bit5
//     PlcTask Outputs/G_IO.arDO[29]/Ch[6] <-> DO1/0016ETP Output-bit maping/Digital output CH1-bit6
//     PlcTask Outputs/G_IO.arDO[29]/Ch[7] <-> DO1/0016ETP Output-bit maping/Digital output CH1-bit7
//     PlcTask Outputs/G_IO.arDO[29]/Ch[8] <-> DO1/0016ETP Output-bit maping/Digital output CH2-bit0
//     PlcTask Outputs/G_IO.arDO[29]/Ch[9] <-> DO1/0016ETP Output-bit maping/Digital output CH2-bit1
//   kittingDeca/kittingDeca Instance <-> rem_wf/rem7_valve
//     PlcTask Outputs/G_IO.arDO[30]/Ch[0] <-> Module 1 (C2S-EC-24B)/Outputs/valve[1..4][0]
//     PlcTask Outputs/G_IO.arDO[30]/Ch[10] <-> Module 1 (C2S-EC-24B)/Outputs/valve[5..8][2]
//     PlcTask Outputs/G_IO.arDO[30]/Ch[11] <-> Module 1 (C2S-EC-24B)/Outputs/valve[5..8][3]
//     PlcTask Outputs/G_IO.arDO[30]/Ch[12] <-> Module 1 (C2S-EC-24B)/Outputs/valve[5..8][4]
//     PlcTask Outputs/G_IO.arDO[30]/Ch[13] <-> Module 1 (C2S-EC-24B)/Outputs/valve[5..8][5]
//     PlcTask Outputs/G_IO.arDO[30]/Ch[14] <-> Module 1 (C2S-EC-24B)/Outputs/valve[5..8][6]
//     PlcTask Outputs/G_IO.arDO[30]/Ch[15] <-> Module 1 (C2S-EC-24B)/Outputs/valve[5..8][7]
//     PlcTask Outputs/G_IO.arDO[30]/Ch[1] <-> Module 1 (C2S-EC-24B)/Outputs/valve[1..4][1]
//     PlcTask Outputs/G_IO.arDO[30]/Ch[2] <-> Module 1 (C2S-EC-24B)/Outputs/valve[1..4][2]
//     PlcTask Outputs/G_IO.arDO[30]/Ch[3] <-> Module 1 (C2S-EC-24B)/Outputs/valve[1..4][3]
//     PlcTask Outputs/G_IO.arDO[30]/Ch[4] <-> Module 1 (C2S-EC-24B)/Outputs/valve[1..4][4]
//     PlcTask Outputs/G_IO.arDO[30]/Ch[5] <-> Module 1 (C2S-EC-24B)/Outputs/valve[1..4][5]
//     PlcTask Outputs/G_IO.arDO[30]/Ch[6] <-> Module 1 (C2S-EC-24B)/Outputs/valve[1..4][6]
//     PlcTask Outputs/G_IO.arDO[30]/Ch[7] <-> Module 1 (C2S-EC-24B)/Outputs/valve[1..4][7]
//     PlcTask Outputs/G_IO.arDO[30]/Ch[8] <-> Module 1 (C2S-EC-24B)/Outputs/valve[5..8][0]
//     PlcTask Outputs/G_IO.arDO[30]/Ch[9] <-> Module 1 (C2S-EC-24B)/Outputs/valve[5..8][1]
//     PlcTask Outputs/G_IO.arDO[31]/Ch[0] <-> Module 1 (C2S-EC-24B)/Outputs/valve[9..12][0]
//     PlcTask Outputs/G_IO.arDO[31]/Ch[1] <-> Module 1 (C2S-EC-24B)/Outputs/valve[9..12][1]
//     PlcTask Outputs/G_IO.arDO[31]/Ch[2] <-> Module 1 (C2S-EC-24B)/Outputs/valve[9..12][2]
//     PlcTask Outputs/G_IO.arDO[31]/Ch[3] <-> Module 1 (C2S-EC-24B)/Outputs/valve[9..12][3]
//     PlcTask Outputs/G_IO.arDO[31]/Ch[4] <-> Module 1 (C2S-EC-24B)/Outputs/valve[9..12][4]
//     PlcTask Outputs/G_IO.arDO[31]/Ch[5] <-> Module 1 (C2S-EC-24B)/Outputs/valve[9..12][5]
//     PlcTask Outputs/G_IO.arDO[31]/Ch[6] <-> Module 1 (C2S-EC-24B)/Outputs/valve[9..12][6]
//     PlcTask Outputs/G_IO.arDO[31]/Ch[7] <-> Module 1 (C2S-EC-24B)/Outputs/valve[9..12][7]
//   kittingDeca/kittingDeca Instance <-> rem_wf/rem8_dio
//     PlcTask Inputs/G_IO.arDI[32]/Ch[0] <-> DI0/1600END input-bit maping/Digital input CH1-bit0
//     PlcTask Inputs/G_IO.arDI[32]/Ch[10] <-> DI0/1600END input-bit maping/Digital input CH2-bit2
//     PlcTask Inputs/G_IO.arDI[32]/Ch[11] <-> DI0/1600END input-bit maping/Digital input CH2-bit3
//     PlcTask Inputs/G_IO.arDI[32]/Ch[12] <-> DI0/1600END input-bit maping/Digital input CH2-bit4
//     PlcTask Inputs/G_IO.arDI[32]/Ch[13] <-> DI0/1600END input-bit maping/Digital input CH2-bit5
//     PlcTask Inputs/G_IO.arDI[32]/Ch[14] <-> DI0/1600END input-bit maping/Digital input CH2-bit6
//     PlcTask Inputs/G_IO.arDI[32]/Ch[15] <-> DI0/1600END input-bit maping/Digital input CH2-bit7
//     PlcTask Inputs/G_IO.arDI[32]/Ch[1] <-> DI0/1600END input-bit maping/Digital input CH1-bit1
//     PlcTask Inputs/G_IO.arDI[32]/Ch[2] <-> DI0/1600END input-bit maping/Digital input CH1-bit2
//     PlcTask Inputs/G_IO.arDI[32]/Ch[3] <-> DI0/1600END input-bit maping/Digital input CH1-bit3
//     PlcTask Inputs/G_IO.arDI[32]/Ch[4] <-> DI0/1600END input-bit maping/Digital input CH1-bit4
//     PlcTask Inputs/G_IO.arDI[32]/Ch[5] <-> DI0/1600END input-bit maping/Digital input CH1-bit5
//     PlcTask Inputs/G_IO.arDI[32]/Ch[6] <-> DI0/1600END input-bit maping/Digital input CH1-bit6
//     PlcTask Inputs/G_IO.arDI[32]/Ch[7] <-> DI0/1600END input-bit maping/Digital input CH1-bit7
//     PlcTask Inputs/G_IO.arDI[32]/Ch[8] <-> DI0/1600END input-bit maping/Digital input CH2-bit0
//     PlcTask Inputs/G_IO.arDI[32]/Ch[9] <-> DI0/1600END input-bit maping/Digital input CH2-bit1
//     PlcTask Inputs/G_IO.arDI[33]/Ch[0] <-> DI1/1600END input-bit maping/Digital input CH1-bit0
//     PlcTask Inputs/G_IO.arDI[33]/Ch[10] <-> DI1/1600END input-bit maping/Digital input CH2-bit2
//     PlcTask Inputs/G_IO.arDI[33]/Ch[11] <-> DI1/1600END input-bit maping/Digital input CH2-bit3
//     PlcTask Inputs/G_IO.arDI[33]/Ch[12] <-> DI1/1600END input-bit maping/Digital input CH2-bit4
//     PlcTask Inputs/G_IO.arDI[33]/Ch[13] <-> DI1/1600END input-bit maping/Digital input CH2-bit5
//     PlcTask Inputs/G_IO.arDI[33]/Ch[14] <-> DI1/1600END input-bit maping/Digital input CH2-bit6
//     PlcTask Inputs/G_IO.arDI[33]/Ch[15] <-> DI1/1600END input-bit maping/Digital input CH2-bit7
//     PlcTask Inputs/G_IO.arDI[33]/Ch[1] <-> DI1/1600END input-bit maping/Digital input CH1-bit1
//     PlcTask Inputs/G_IO.arDI[33]/Ch[2] <-> DI1/1600END input-bit maping/Digital input CH1-bit2
//     PlcTask Inputs/G_IO.arDI[33]/Ch[3] <-> DI1/1600END input-bit maping/Digital input CH1-bit3
//     PlcTask Inputs/G_IO.arDI[33]/Ch[4] <-> DI1/1600END input-bit maping/Digital input CH1-bit4
//     PlcTask Inputs/G_IO.arDI[33]/Ch[5] <-> DI1/1600END input-bit maping/Digital input CH1-bit5
//     PlcTask Inputs/G_IO.arDI[33]/Ch[6] <-> DI1/1600END input-bit maping/Digital input CH1-bit6
//     PlcTask Inputs/G_IO.arDI[33]/Ch[7] <-> DI1/1600END input-bit maping/Digital input CH1-bit7
//     PlcTask Inputs/G_IO.arDI[33]/Ch[8] <-> DI1/1600END input-bit maping/Digital input CH2-bit0
//     PlcTask Inputs/G_IO.arDI[33]/Ch[9] <-> DI1/1600END input-bit maping/Digital input CH2-bit1
//     PlcTask Inputs/G_IO.arDI[34]/Ch[0] <-> DI2/1600END input-bit maping/Digital input CH1-bit0
//     PlcTask Inputs/G_IO.arDI[34]/Ch[10] <-> DI2/1600END input-bit maping/Digital input CH2-bit2
//     PlcTask Inputs/G_IO.arDI[34]/Ch[11] <-> DI2/1600END input-bit maping/Digital input CH2-bit3
//     PlcTask Inputs/G_IO.arDI[34]/Ch[12] <-> DI2/1600END input-bit maping/Digital input CH2-bit4
//     PlcTask Inputs/G_IO.arDI[34]/Ch[13] <-> DI2/1600END input-bit maping/Digital input CH2-bit5
//     PlcTask Inputs/G_IO.arDI[34]/Ch[14] <-> DI2/1600END input-bit maping/Digital input CH2-bit6
//     PlcTask Inputs/G_IO.arDI[34]/Ch[15] <-> DI2/1600END input-bit maping/Digital input CH2-bit7
//     PlcTask Inputs/G_IO.arDI[34]/Ch[1] <-> DI2/1600END input-bit maping/Digital input CH1-bit1
//     PlcTask Inputs/G_IO.arDI[34]/Ch[2] <-> DI2/1600END input-bit maping/Digital input CH1-bit2
//     PlcTask Inputs/G_IO.arDI[34]/Ch[3] <-> DI2/1600END input-bit maping/Digital input CH1-bit3
//     PlcTask Inputs/G_IO.arDI[34]/Ch[4] <-> DI2/1600END input-bit maping/Digital input CH1-bit4
//     PlcTask Inputs/G_IO.arDI[34]/Ch[5] <-> DI2/1600END input-bit maping/Digital input CH1-bit5
//     PlcTask Inputs/G_IO.arDI[34]/Ch[6] <-> DI2/1600END input-bit maping/Digital input CH1-bit6
//     PlcTask Inputs/G_IO.arDI[34]/Ch[7] <-> DI2/1600END input-bit maping/Digital input CH1-bit7
//     PlcTask Inputs/G_IO.arDI[34]/Ch[8] <-> DI2/1600END input-bit maping/Digital input CH2-bit0
//     PlcTask Inputs/G_IO.arDI[34]/Ch[9] <-> DI2/1600END input-bit maping/Digital input CH2-bit1
//     PlcTask Inputs/G_IO.arDI[35]/Ch[0] <-> DI3/1600END input-bit maping/Digital input CH1-bit0
//     PlcTask Inputs/G_IO.arDI[35]/Ch[10] <-> DI3/1600END input-bit maping/Digital input CH2-bit2
//     PlcTask Inputs/G_IO.arDI[35]/Ch[11] <-> DI3/1600END input-bit maping/Digital input CH2-bit3
//     PlcTask Inputs/G_IO.arDI[35]/Ch[12] <-> DI3/1600END input-bit maping/Digital input CH2-bit4
//     PlcTask Inputs/G_IO.arDI[35]/Ch[13] <-> DI3/1600END input-bit maping/Digital input CH2-bit5
//     PlcTask Inputs/G_IO.arDI[35]/Ch[14] <-> DI3/1600END input-bit maping/Digital input CH2-bit6
//     PlcTask Inputs/G_IO.arDI[35]/Ch[15] <-> DI3/1600END input-bit maping/Digital input CH2-bit7
//     PlcTask Inputs/G_IO.arDI[35]/Ch[1] <-> DI3/1600END input-bit maping/Digital input CH1-bit1
//     PlcTask Inputs/G_IO.arDI[35]/Ch[2] <-> DI3/1600END input-bit maping/Digital input CH1-bit2
//     PlcTask Inputs/G_IO.arDI[35]/Ch[3] <-> DI3/1600END input-bit maping/Digital input CH1-bit3
//     PlcTask Inputs/G_IO.arDI[35]/Ch[4] <-> DI3/1600END input-bit maping/Digital input CH1-bit4
//     PlcTask Inputs/G_IO.arDI[35]/Ch[5] <-> DI3/1600END input-bit maping/Digital input CH1-bit5
//     PlcTask Inputs/G_IO.arDI[35]/Ch[6] <-> DI3/1600END input-bit maping/Digital input CH1-bit6
//     PlcTask Inputs/G_IO.arDI[35]/Ch[7] <-> DI3/1600END input-bit maping/Digital input CH1-bit7
//     PlcTask Inputs/G_IO.arDI[35]/Ch[8] <-> DI3/1600END input-bit maping/Digital input CH2-bit0
//     PlcTask Inputs/G_IO.arDI[35]/Ch[9] <-> DI3/1600END input-bit maping/Digital input CH2-bit1
//     PlcTask Outputs/G_IO.arDO[32]/Ch[0] <-> DO0/0016ETP Output-bit maping/Digital output CH1-bit0
//     PlcTask Outputs/G_IO.arDO[32]/Ch[10] <-> DO0/0016ETP Output-bit maping/Digital output CH2-bit2
//     PlcTask Outputs/G_IO.arDO[32]/Ch[11] <-> DO0/0016ETP Output-bit maping/Digital output CH2-bit3
//     PlcTask Outputs/G_IO.arDO[32]/Ch[12] <-> DO0/0016ETP Output-bit maping/Digital output CH2-bit4
//     PlcTask Outputs/G_IO.arDO[32]/Ch[13] <-> DO0/0016ETP Output-bit maping/Digital output CH2-bit5
//     PlcTask Outputs/G_IO.arDO[32]/Ch[14] <-> DO0/0016ETP Output-bit maping/Digital output CH2-bit6
//     PlcTask Outputs/G_IO.arDO[32]/Ch[15] <-> DO0/0016ETP Output-bit maping/Digital output CH2-bit7
//     PlcTask Outputs/G_IO.arDO[32]/Ch[1] <-> DO0/0016ETP Output-bit maping/Digital output CH1-bit1
//     PlcTask Outputs/G_IO.arDO[32]/Ch[2] <-> DO0/0016ETP Output-bit maping/Digital output CH1-bit2
//     PlcTask Outputs/G_IO.arDO[32]/Ch[3] <-> DO0/0016ETP Output-bit maping/Digital output CH1-bit3
//     PlcTask Outputs/G_IO.arDO[32]/Ch[4] <-> DO0/0016ETP Output-bit maping/Digital output CH1-bit4
//     PlcTask Outputs/G_IO.arDO[32]/Ch[5] <-> DO0/0016ETP Output-bit maping/Digital output CH1-bit5
//     PlcTask Outputs/G_IO.arDO[32]/Ch[6] <-> DO0/0016ETP Output-bit maping/Digital output CH1-bit6
//     PlcTask Outputs/G_IO.arDO[32]/Ch[7] <-> DO0/0016ETP Output-bit maping/Digital output CH1-bit7
//     PlcTask Outputs/G_IO.arDO[32]/Ch[8] <-> DO0/0016ETP Output-bit maping/Digital output CH2-bit0
//     PlcTask Outputs/G_IO.arDO[32]/Ch[9] <-> DO0/0016ETP Output-bit maping/Digital output CH2-bit1
//     PlcTask Outputs/G_IO.arDO[33]/Ch[0] <-> DO1/0016ETP Output-bit maping/Digital output CH1-bit0
//     PlcTask Outputs/G_IO.arDO[33]/Ch[10] <-> DO1/0016ETP Output-bit maping/Digital output CH2-bit2
//     PlcTask Outputs/G_IO.arDO[33]/Ch[11] <-> DO1/0016ETP Output-bit maping/Digital output CH2-bit3
//     PlcTask Outputs/G_IO.arDO[33]/Ch[12] <-> DO1/0016ETP Output-bit maping/Digital output CH2-bit4
//     PlcTask Outputs/G_IO.arDO[33]/Ch[13] <-> DO1/0016ETP Output-bit maping/Digital output CH2-bit5
//     PlcTask Outputs/G_IO.arDO[33]/Ch[14] <-> DO1/0016ETP Output-bit maping/Digital output CH2-bit6
//     PlcTask Outputs/G_IO.arDO[33]/Ch[15] <-> DO1/0016ETP Output-bit maping/Digital output CH2-bit7
//     PlcTask Outputs/G_IO.arDO[33]/Ch[1] <-> DO1/0016ETP Output-bit maping/Digital output CH1-bit1
//     PlcTask Outputs/G_IO.arDO[33]/Ch[2] <-> DO1/0016ETP Output-bit maping/Digital output CH1-bit2
//     PlcTask Outputs/G_IO.arDO[33]/Ch[3] <-> DO1/0016ETP Output-bit maping/Digital output CH1-bit3
//     PlcTask Outputs/G_IO.arDO[33]/Ch[4] <-> DO1/0016ETP Output-bit maping/Digital output CH1-bit4
//     PlcTask Outputs/G_IO.arDO[33]/Ch[5] <-> DO1/0016ETP Output-bit maping/Digital output CH1-bit5
//     PlcTask Outputs/G_IO.arDO[33]/Ch[6] <-> DO1/0016ETP Output-bit maping/Digital output CH1-bit6
//     PlcTask Outputs/G_IO.arDO[33]/Ch[7] <-> DO1/0016ETP Output-bit maping/Digital output CH1-bit7
//     PlcTask Outputs/G_IO.arDO[33]/Ch[8] <-> DO1/0016ETP Output-bit maping/Digital output CH2-bit0
//     PlcTask Outputs/G_IO.arDO[33]/Ch[9] <-> DO1/0016ETP Output-bit maping/Digital output CH2-bit1
//   kittingDeca/kittingDeca Instance <-> rem_wf/rem8_valve
//     PlcTask Outputs/G_IO.arDO[34]/Ch[0] <-> Module 1 (C2S-EC-24B)/Outputs/valve[1..4][0]
//     PlcTask Outputs/G_IO.arDO[34]/Ch[10] <-> Module 1 (C2S-EC-24B)/Outputs/valve[5..8][2]
//     PlcTask Outputs/G_IO.arDO[34]/Ch[11] <-> Module 1 (C2S-EC-24B)/Outputs/valve[5..8][3]
//     PlcTask Outputs/G_IO.arDO[34]/Ch[12] <-> Module 1 (C2S-EC-24B)/Outputs/valve[5..8][4]
//     PlcTask Outputs/G_IO.arDO[34]/Ch[13] <-> Module 1 (C2S-EC-24B)/Outputs/valve[5..8][5]
//     PlcTask Outputs/G_IO.arDO[34]/Ch[14] <-> Module 1 (C2S-EC-24B)/Outputs/valve[5..8][6]
//     PlcTask Outputs/G_IO.arDO[34]/Ch[15] <-> Module 1 (C2S-EC-24B)/Outputs/valve[5..8][7]
//     PlcTask Outputs/G_IO.arDO[34]/Ch[1] <-> Module 1 (C2S-EC-24B)/Outputs/valve[1..4][1]
//     PlcTask Outputs/G_IO.arDO[34]/Ch[2] <-> Module 1 (C2S-EC-24B)/Outputs/valve[1..4][2]
//     PlcTask Outputs/G_IO.arDO[34]/Ch[3] <-> Module 1 (C2S-EC-24B)/Outputs/valve[1..4][3]
//     PlcTask Outputs/G_IO.arDO[34]/Ch[4] <-> Module 1 (C2S-EC-24B)/Outputs/valve[1..4][4]
//     PlcTask Outputs/G_IO.arDO[34]/Ch[5] <-> Module 1 (C2S-EC-24B)/Outputs/valve[1..4][5]
//     PlcTask Outputs/G_IO.arDO[34]/Ch[6] <-> Module 1 (C2S-EC-24B)/Outputs/valve[1..4][6]
//     PlcTask Outputs/G_IO.arDO[34]/Ch[7] <-> Module 1 (C2S-EC-24B)/Outputs/valve[1..4][7]
//     PlcTask Outputs/G_IO.arDO[34]/Ch[8] <-> Module 1 (C2S-EC-24B)/Outputs/valve[5..8][0]
//     PlcTask Outputs/G_IO.arDO[34]/Ch[9] <-> Module 1 (C2S-EC-24B)/Outputs/valve[5..8][1]
//     PlcTask Outputs/G_IO.arDO[35]/Ch[0] <-> Module 1 (C2S-EC-24B)/Outputs/valve[9..12][0]
//     PlcTask Outputs/G_IO.arDO[35]/Ch[1] <-> Module 1 (C2S-EC-24B)/Outputs/valve[9..12][1]
//     PlcTask Outputs/G_IO.arDO[35]/Ch[2] <-> Module 1 (C2S-EC-24B)/Outputs/valve[9..12][2]
//     PlcTask Outputs/G_IO.arDO[35]/Ch[3] <-> Module 1 (C2S-EC-24B)/Outputs/valve[9..12][3]
//     PlcTask Outputs/G_IO.arDO[35]/Ch[4] <-> Module 1 (C2S-EC-24B)/Outputs/valve[9..12][4]
//     PlcTask Outputs/G_IO.arDO[35]/Ch[5] <-> Module 1 (C2S-EC-24B)/Outputs/valve[9..12][5]
//     PlcTask Outputs/G_IO.arDO[35]/Ch[6] <-> Module 1 (C2S-EC-24B)/Outputs/valve[9..12][6]
//     PlcTask Outputs/G_IO.arDO[35]/Ch[7] <-> Module 1 (C2S-EC-24B)/Outputs/valve[9..12][7]
//   kittingDeca/kittingDeca Instance <-> rem_wf/rem9_dio
//     PlcTask Inputs/G_IO.arDI[36]/Ch[0] <-> DI0/1600END input-bit maping/Digital input CH1-bit0
//     PlcTask Inputs/G_IO.arDI[36]/Ch[10] <-> DI0/1600END input-bit maping/Digital input CH2-bit2
//     PlcTask Inputs/G_IO.arDI[36]/Ch[11] <-> DI0/1600END input-bit maping/Digital input CH2-bit3
//     PlcTask Inputs/G_IO.arDI[36]/Ch[12] <-> DI0/1600END input-bit maping/Digital input CH2-bit4
//     PlcTask Inputs/G_IO.arDI[36]/Ch[13] <-> DI0/1600END input-bit maping/Digital input CH2-bit5
//     PlcTask Inputs/G_IO.arDI[36]/Ch[14] <-> DI0/1600END input-bit maping/Digital input CH2-bit6
//     PlcTask Inputs/G_IO.arDI[36]/Ch[15] <-> DI0/1600END input-bit maping/Digital input CH2-bit7
//     PlcTask Inputs/G_IO.arDI[36]/Ch[1] <-> DI0/1600END input-bit maping/Digital input CH1-bit1
//     PlcTask Inputs/G_IO.arDI[36]/Ch[2] <-> DI0/1600END input-bit maping/Digital input CH1-bit2
//     PlcTask Inputs/G_IO.arDI[36]/Ch[3] <-> DI0/1600END input-bit maping/Digital input CH1-bit3
//     PlcTask Inputs/G_IO.arDI[36]/Ch[4] <-> DI0/1600END input-bit maping/Digital input CH1-bit4
//     PlcTask Inputs/G_IO.arDI[36]/Ch[5] <-> DI0/1600END input-bit maping/Digital input CH1-bit5
//     PlcTask Inputs/G_IO.arDI[36]/Ch[6] <-> DI0/1600END input-bit maping/Digital input CH1-bit6
//     PlcTask Inputs/G_IO.arDI[36]/Ch[7] <-> DI0/1600END input-bit maping/Digital input CH1-bit7
//     PlcTask Inputs/G_IO.arDI[36]/Ch[8] <-> DI0/1600END input-bit maping/Digital input CH2-bit0
//     PlcTask Inputs/G_IO.arDI[36]/Ch[9] <-> DI0/1600END input-bit maping/Digital input CH2-bit1
//     PlcTask Inputs/G_IO.arDI[37]/Ch[0] <-> DI1/1600END input-bit maping/Digital input CH1-bit0
//     PlcTask Inputs/G_IO.arDI[37]/Ch[10] <-> DI1/1600END input-bit maping/Digital input CH2-bit2
//     PlcTask Inputs/G_IO.arDI[37]/Ch[11] <-> DI1/1600END input-bit maping/Digital input CH2-bit3
//     PlcTask Inputs/G_IO.arDI[37]/Ch[12] <-> DI1/1600END input-bit maping/Digital input CH2-bit4
//     PlcTask Inputs/G_IO.arDI[37]/Ch[13] <-> DI1/1600END input-bit maping/Digital input CH2-bit5
//     PlcTask Inputs/G_IO.arDI[37]/Ch[14] <-> DI1/1600END input-bit maping/Digital input CH2-bit6
//     PlcTask Inputs/G_IO.arDI[37]/Ch[15] <-> DI1/1600END input-bit maping/Digital input CH2-bit7
//     PlcTask Inputs/G_IO.arDI[37]/Ch[1] <-> DI1/1600END input-bit maping/Digital input CH1-bit1
//     PlcTask Inputs/G_IO.arDI[37]/Ch[2] <-> DI1/1600END input-bit maping/Digital input CH1-bit2
//     PlcTask Inputs/G_IO.arDI[37]/Ch[3] <-> DI1/1600END input-bit maping/Digital input CH1-bit3
//     PlcTask Inputs/G_IO.arDI[37]/Ch[4] <-> DI1/1600END input-bit maping/Digital input CH1-bit4
//     PlcTask Inputs/G_IO.arDI[37]/Ch[5] <-> DI1/1600END input-bit maping/Digital input CH1-bit5
//     PlcTask Inputs/G_IO.arDI[37]/Ch[6] <-> DI1/1600END input-bit maping/Digital input CH1-bit6
//     PlcTask Inputs/G_IO.arDI[37]/Ch[7] <-> DI1/1600END input-bit maping/Digital input CH1-bit7
//     PlcTask Inputs/G_IO.arDI[37]/Ch[8] <-> DI1/1600END input-bit maping/Digital input CH2-bit0
//     PlcTask Inputs/G_IO.arDI[37]/Ch[9] <-> DI1/1600END input-bit maping/Digital input CH2-bit1
//     PlcTask Inputs/G_IO.arDI[38]/Ch[0] <-> DI2/1600END input-bit maping/Digital input CH1-bit0
//     PlcTask Inputs/G_IO.arDI[38]/Ch[10] <-> DI2/1600END input-bit maping/Digital input CH2-bit2
//     PlcTask Inputs/G_IO.arDI[38]/Ch[11] <-> DI2/1600END input-bit maping/Digital input CH2-bit3
//     PlcTask Inputs/G_IO.arDI[38]/Ch[12] <-> DI2/1600END input-bit maping/Digital input CH2-bit4
//     PlcTask Inputs/G_IO.arDI[38]/Ch[13] <-> DI2/1600END input-bit maping/Digital input CH2-bit5
//     PlcTask Inputs/G_IO.arDI[38]/Ch[14] <-> DI2/1600END input-bit maping/Digital input CH2-bit6
//     PlcTask Inputs/G_IO.arDI[38]/Ch[15] <-> DI2/1600END input-bit maping/Digital input CH2-bit7
//     PlcTask Inputs/G_IO.arDI[38]/Ch[1] <-> DI2/1600END input-bit maping/Digital input CH1-bit1
//     PlcTask Inputs/G_IO.arDI[38]/Ch[2] <-> DI2/1600END input-bit maping/Digital input CH1-bit2
//     PlcTask Inputs/G_IO.arDI[38]/Ch[3] <-> DI2/1600END input-bit maping/Digital input CH1-bit3
//     PlcTask Inputs/G_IO.arDI[38]/Ch[4] <-> DI2/1600END input-bit maping/Digital input CH1-bit4
//     PlcTask Inputs/G_IO.arDI[38]/Ch[5] <-> DI2/1600END input-bit maping/Digital input CH1-bit5
//     PlcTask Inputs/G_IO.arDI[38]/Ch[6] <-> DI2/1600END input-bit maping/Digital input CH1-bit6
//     PlcTask Inputs/G_IO.arDI[38]/Ch[7] <-> DI2/1600END input-bit maping/Digital input CH1-bit7
//     PlcTask Inputs/G_IO.arDI[38]/Ch[8] <-> DI2/1600END input-bit maping/Digital input CH2-bit0
//     PlcTask Inputs/G_IO.arDI[38]/Ch[9] <-> DI2/1600END input-bit maping/Digital input CH2-bit1
//     PlcTask Inputs/G_IO.arDI[39]/Ch[0] <-> DI3/1600END input-bit maping/Digital input CH1-bit0
//     PlcTask Inputs/G_IO.arDI[39]/Ch[10] <-> DI3/1600END input-bit maping/Digital input CH2-bit2
//     PlcTask Inputs/G_IO.arDI[39]/Ch[11] <-> DI3/1600END input-bit maping/Digital input CH2-bit3
//     PlcTask Inputs/G_IO.arDI[39]/Ch[12] <-> DI3/1600END input-bit maping/Digital input CH2-bit4
//     PlcTask Inputs/G_IO.arDI[39]/Ch[13] <-> DI3/1600END input-bit maping/Digital input CH2-bit5
//     PlcTask Inputs/G_IO.arDI[39]/Ch[14] <-> DI3/1600END input-bit maping/Digital input CH2-bit6
//     PlcTask Inputs/G_IO.arDI[39]/Ch[15] <-> DI3/1600END input-bit maping/Digital input CH2-bit7
//     PlcTask Inputs/G_IO.arDI[39]/Ch[1] <-> DI3/1600END input-bit maping/Digital input CH1-bit1
//     PlcTask Inputs/G_IO.arDI[39]/Ch[2] <-> DI3/1600END input-bit maping/Digital input CH1-bit2
//     PlcTask Inputs/G_IO.arDI[39]/Ch[3] <-> DI3/1600END input-bit maping/Digital input CH1-bit3
//     PlcTask Inputs/G_IO.arDI[39]/Ch[4] <-> DI3/1600END input-bit maping/Digital input CH1-bit4
//     PlcTask Inputs/G_IO.arDI[39]/Ch[5] <-> DI3/1600END input-bit maping/Digital input CH1-bit5
//     PlcTask Inputs/G_IO.arDI[39]/Ch[6] <-> DI3/1600END input-bit maping/Digital input CH1-bit6
//     PlcTask Inputs/G_IO.arDI[39]/Ch[7] <-> DI3/1600END input-bit maping/Digital input CH1-bit7
//     PlcTask Inputs/G_IO.arDI[39]/Ch[8] <-> DI3/1600END input-bit maping/Digital input CH2-bit0
//     PlcTask Inputs/G_IO.arDI[39]/Ch[9] <-> DI3/1600END input-bit maping/Digital input CH2-bit1
//     PlcTask Outputs/G_IO.arDO[36]/Ch[0] <-> DO0/0016ETP Output-bit maping/Digital output CH1-bit0
//     PlcTask Outputs/G_IO.arDO[36]/Ch[10] <-> DO0/0016ETP Output-bit maping/Digital output CH2-bit2
//     PlcTask Outputs/G_IO.arDO[36]/Ch[11] <-> DO0/0016ETP Output-bit maping/Digital output CH2-bit3
//     PlcTask Outputs/G_IO.arDO[36]/Ch[12] <-> DO0/0016ETP Output-bit maping/Digital output CH2-bit4
//     PlcTask Outputs/G_IO.arDO[36]/Ch[13] <-> DO0/0016ETP Output-bit maping/Digital output CH2-bit5
//     PlcTask Outputs/G_IO.arDO[36]/Ch[14] <-> DO0/0016ETP Output-bit maping/Digital output CH2-bit6
//     PlcTask Outputs/G_IO.arDO[36]/Ch[15] <-> DO0/0016ETP Output-bit maping/Digital output CH2-bit7
//     PlcTask Outputs/G_IO.arDO[36]/Ch[1] <-> DO0/0016ETP Output-bit maping/Digital output CH1-bit1
//     PlcTask Outputs/G_IO.arDO[36]/Ch[2] <-> DO0/0016ETP Output-bit maping/Digital output CH1-bit2
//     PlcTask Outputs/G_IO.arDO[36]/Ch[3] <-> DO0/0016ETP Output-bit maping/Digital output CH1-bit3
//     PlcTask Outputs/G_IO.arDO[36]/Ch[4] <-> DO0/0016ETP Output-bit maping/Digital output CH1-bit4
//     PlcTask Outputs/G_IO.arDO[36]/Ch[5] <-> DO0/0016ETP Output-bit maping/Digital output CH1-bit5
//     PlcTask Outputs/G_IO.arDO[36]/Ch[6] <-> DO0/0016ETP Output-bit maping/Digital output CH1-bit6
//     PlcTask Outputs/G_IO.arDO[36]/Ch[7] <-> DO0/0016ETP Output-bit maping/Digital output CH1-bit7
//     PlcTask Outputs/G_IO.arDO[36]/Ch[8] <-> DO0/0016ETP Output-bit maping/Digital output CH2-bit0
//     PlcTask Outputs/G_IO.arDO[36]/Ch[9] <-> DO0/0016ETP Output-bit maping/Digital output CH2-bit1
//     PlcTask Outputs/G_IO.arDO[37]/Ch[0] <-> DO1/0016ETP Output-bit maping/Digital output CH1-bit0
//     PlcTask Outputs/G_IO.arDO[37]/Ch[10] <-> DO1/0016ETP Output-bit maping/Digital output CH2-bit2
//     PlcTask Outputs/G_IO.arDO[37]/Ch[11] <-> DO1/0016ETP Output-bit maping/Digital output CH2-bit3
//     PlcTask Outputs/G_IO.arDO[37]/Ch[12] <-> DO1/0016ETP Output-bit maping/Digital output CH2-bit4
//     PlcTask Outputs/G_IO.arDO[37]/Ch[13] <-> DO1/0016ETP Output-bit maping/Digital output CH2-bit5
//     PlcTask Outputs/G_IO.arDO[37]/Ch[14] <-> DO1/0016ETP Output-bit maping/Digital output CH2-bit6
//     PlcTask Outputs/G_IO.arDO[37]/Ch[15] <-> DO1/0016ETP Output-bit maping/Digital output CH2-bit7
//     PlcTask Outputs/G_IO.arDO[37]/Ch[1] <-> DO1/0016ETP Output-bit maping/Digital output CH1-bit1
//     PlcTask Outputs/G_IO.arDO[37]/Ch[2] <-> DO1/0016ETP Output-bit maping/Digital output CH1-bit2
//     PlcTask Outputs/G_IO.arDO[37]/Ch[3] <-> DO1/0016ETP Output-bit maping/Digital output CH1-bit3
//     PlcTask Outputs/G_IO.arDO[37]/Ch[4] <-> DO1/0016ETP Output-bit maping/Digital output CH1-bit4
//     PlcTask Outputs/G_IO.arDO[37]/Ch[5] <-> DO1/0016ETP Output-bit maping/Digital output CH1-bit5
//     PlcTask Outputs/G_IO.arDO[37]/Ch[6] <-> DO1/0016ETP Output-bit maping/Digital output CH1-bit6
//     PlcTask Outputs/G_IO.arDO[37]/Ch[7] <-> DO1/0016ETP Output-bit maping/Digital output CH1-bit7
//     PlcTask Outputs/G_IO.arDO[37]/Ch[8] <-> DO1/0016ETP Output-bit maping/Digital output CH2-bit0
//     PlcTask Outputs/G_IO.arDO[37]/Ch[9] <-> DO1/0016ETP Output-bit maping/Digital output CH2-bit1
//   kittingDeca/kittingDeca Instance <-> rem_wf/rem9_valve
//     PlcTask Outputs/G_IO.arDO[38]/Ch[0] <-> Module 1 (C2S-EC-24B)/Outputs/valve[1..4][0]
//     PlcTask Outputs/G_IO.arDO[38]/Ch[10] <-> Module 1 (C2S-EC-24B)/Outputs/valve[5..8][2]
//     PlcTask Outputs/G_IO.arDO[38]/Ch[11] <-> Module 1 (C2S-EC-24B)/Outputs/valve[5..8][3]
//     PlcTask Outputs/G_IO.arDO[38]/Ch[12] <-> Module 1 (C2S-EC-24B)/Outputs/valve[5..8][4]
//     PlcTask Outputs/G_IO.arDO[38]/Ch[13] <-> Module 1 (C2S-EC-24B)/Outputs/valve[5..8][5]
//     PlcTask Outputs/G_IO.arDO[38]/Ch[14] <-> Module 1 (C2S-EC-24B)/Outputs/valve[5..8][6]
//     PlcTask Outputs/G_IO.arDO[38]/Ch[15] <-> Module 1 (C2S-EC-24B)/Outputs/valve[5..8][7]
//     PlcTask Outputs/G_IO.arDO[38]/Ch[1] <-> Module 1 (C2S-EC-24B)/Outputs/valve[1..4][1]
//     PlcTask Outputs/G_IO.arDO[38]/Ch[2] <-> Module 1 (C2S-EC-24B)/Outputs/valve[1..4][2]
//     PlcTask Outputs/G_IO.arDO[38]/Ch[3] <-> Module 1 (C2S-EC-24B)/Outputs/valve[1..4][3]
//     PlcTask Outputs/G_IO.arDO[38]/Ch[4] <-> Module 1 (C2S-EC-24B)/Outputs/valve[1..4][4]
//     PlcTask Outputs/G_IO.arDO[38]/Ch[5] <-> Module 1 (C2S-EC-24B)/Outputs/valve[1..4][5]
//     PlcTask Outputs/G_IO.arDO[38]/Ch[6] <-> Module 1 (C2S-EC-24B)/Outputs/valve[1..4][6]
//     PlcTask Outputs/G_IO.arDO[38]/Ch[7] <-> Module 1 (C2S-EC-24B)/Outputs/valve[1..4][7]
//     PlcTask Outputs/G_IO.arDO[38]/Ch[8] <-> Module 1 (C2S-EC-24B)/Outputs/valve[5..8][0]
//     PlcTask Outputs/G_IO.arDO[38]/Ch[9] <-> Module 1 (C2S-EC-24B)/Outputs/valve[5..8][1]
//     PlcTask Outputs/G_IO.arDO[39]/Ch[0] <-> Module 1 (C2S-EC-24B)/Outputs/valve[9..12][0]
//     PlcTask Outputs/G_IO.arDO[39]/Ch[1] <-> Module 1 (C2S-EC-24B)/Outputs/valve[9..12][1]
//     PlcTask Outputs/G_IO.arDO[39]/Ch[2] <-> Module 1 (C2S-EC-24B)/Outputs/valve[9..12][2]
//     PlcTask Outputs/G_IO.arDO[39]/Ch[3] <-> Module 1 (C2S-EC-24B)/Outputs/valve[9..12][3]
//     PlcTask Outputs/G_IO.arDO[39]/Ch[4] <-> Module 1 (C2S-EC-24B)/Outputs/valve[9..12][4]
//     PlcTask Outputs/G_IO.arDO[39]/Ch[5] <-> Module 1 (C2S-EC-24B)/Outputs/valve[9..12][5]
//     PlcTask Outputs/G_IO.arDO[39]/Ch[6] <-> Module 1 (C2S-EC-24B)/Outputs/valve[9..12][6]
//     PlcTask Outputs/G_IO.arDO[39]/Ch[7] <-> Module 1 (C2S-EC-24B)/Outputs/valve[9..12][7]
//   kittingDeca/kittingDeca Instance <-> rem_wf/safetyPLC
//     PlcTask Inputs/GVL.safetyin[0] <-> In/In_Dataset1[0]
//     PlcTask Inputs/GVL.safetyin[10] <-> In/In_Dataset2[0]
//     PlcTask Inputs/GVL.safetyin[11] <-> In/In_Dataset2[1]
//     PlcTask Inputs/GVL.safetyin[12] <-> In/In_Dataset2[2]
//     PlcTask Inputs/GVL.safetyin[13] <-> In/In_Dataset2[3]
//     PlcTask Inputs/GVL.safetyin[14] <-> In/In_Dataset2[4]
//     PlcTask Inputs/GVL.safetyin[15] <-> In/In_Dataset2[5]
//     PlcTask Inputs/GVL.safetyin[16] <-> In/In_Dataset2[6]
//     PlcTask Inputs/GVL.safetyin[17] <-> In/In_Dataset2[7]
//     PlcTask Inputs/GVL.safetyin[18] <-> In/In_Dataset2[8]
//     PlcTask Inputs/GVL.safetyin[19] <-> In/In_Dataset2[9]
//     PlcTask Inputs/GVL.safetyin[1] <-> In/In_Dataset1[1]
//     PlcTask Inputs/GVL.safetyin[20] <-> In/In_Dataset3[0]
//     PlcTask Inputs/GVL.safetyin[21] <-> In/In_Dataset3[1]
//     PlcTask Inputs/GVL.safetyin[22] <-> In/In_Dataset3[2]
//     PlcTask Inputs/GVL.safetyin[23] <-> In/In_Dataset3[3]
//     PlcTask Inputs/GVL.safetyin[24] <-> In/In_Dataset3[4]
//     PlcTask Inputs/GVL.safetyin[25] <-> In/In_Dataset3[5]
//     PlcTask Inputs/GVL.safetyin[26] <-> In/In_Dataset3[6]
//     PlcTask Inputs/GVL.safetyin[27] <-> In/In_Dataset3[7]
//     PlcTask Inputs/GVL.safetyin[28] <-> In/In_Dataset3[8]
//     PlcTask Inputs/GVL.safetyin[29] <-> In/In_Dataset3[9]
//     PlcTask Inputs/GVL.safetyin[2] <-> In/In_Dataset1[2]
//     PlcTask Inputs/GVL.safetyin[30] <-> In/In_Dataset4[0]
//     PlcTask Inputs/GVL.safetyin[31] <-> In/In_Dataset4[1]
//     PlcTask Inputs/GVL.safetyin[32] <-> In/In_Dataset4[2]
//     PlcTask Inputs/GVL.safetyin[33] <-> In/In_Dataset4[3]
//     PlcTask Inputs/GVL.safetyin[34] <-> In/In_Dataset4[4]
//     PlcTask Inputs/GVL.safetyin[35] <-> In/In_Dataset4[5]
//     PlcTask Inputs/GVL.safetyin[36] <-> In/In_Dataset4[6]
//     PlcTask Inputs/GVL.safetyin[37] <-> In/In_Dataset4[7]
//     PlcTask Inputs/GVL.safetyin[38] <-> In/In_Dataset4[8]
//     PlcTask Inputs/GVL.safetyin[39] <-> In/In_Dataset4[9]
//     PlcTask Inputs/GVL.safetyin[3] <-> In/In_Dataset1[3]
//     PlcTask Inputs/GVL.safetyin[40] <-> In/In_Dataset5[0]
//     PlcTask Inputs/GVL.safetyin[41] <-> In/In_Dataset5[1]
//     PlcTask Inputs/GVL.safetyin[42] <-> In/In_Dataset5[2]
//     PlcTask Inputs/GVL.safetyin[43] <-> In/In_Dataset5[3]
//     PlcTask Inputs/GVL.safetyin[44] <-> In/In_Dataset5[4]
//     PlcTask Inputs/GVL.safetyin[45] <-> In/In_Dataset5[5]
//     PlcTask Inputs/GVL.safetyin[46] <-> In/In_Dataset5[6]
//     PlcTask Inputs/GVL.safetyin[47] <-> In/In_Dataset5[7]
//     PlcTask Inputs/GVL.safetyin[48] <-> In/In_Dataset5[8]
//     PlcTask Inputs/GVL.safetyin[49] <-> In/In_Dataset5[9]
//     PlcTask Inputs/GVL.safetyin[4] <-> In/In_Dataset1[4]
//     PlcTask Inputs/GVL.safetyin[5] <-> In/In_Dataset1[5]
//     PlcTask Inputs/GVL.safetyin[6] <-> In/In_Dataset1[6]
//     PlcTask Inputs/GVL.safetyin[7] <-> In/In_Dataset1[7]
//     PlcTask Inputs/GVL.safetyin[8] <-> In/In_Dataset1[8]
//     PlcTask Inputs/GVL.safetyin[9] <-> In/In_Dataset1[9]
//     PlcTask Outputs/GVL.safetyOut[0] <-> Out/Out_Dataset1[0]
//     PlcTask Outputs/GVL.safetyOut[10] <-> Out/Out_Dataset2[0]
//     PlcTask Outputs/GVL.safetyOut[11] <-> Out/Out_Dataset2[1]
//     PlcTask Outputs/GVL.safetyOut[12] <-> Out/Out_Dataset2[2]
//     PlcTask Outputs/GVL.safetyOut[13] <-> Out/Out_Dataset2[3]
//     PlcTask Outputs/GVL.safetyOut[14] <-> Out/Out_Dataset2[4]
//     PlcTask Outputs/GVL.safetyOut[15] <-> Out/Out_Dataset2[5]
//     PlcTask Outputs/GVL.safetyOut[16] <-> Out/Out_Dataset2[6]
//     PlcTask Outputs/GVL.safetyOut[17] <-> Out/Out_Dataset2[7]
//     PlcTask Outputs/GVL.safetyOut[18] <-> Out/Out_Dataset2[8]
//     PlcTask Outputs/GVL.safetyOut[19] <-> Out/Out_Dataset2[9]
//     PlcTask Outputs/GVL.safetyOut[1] <-> Out/Out_Dataset1[1]
//     PlcTask Outputs/GVL.safetyOut[20] <-> Out/Out_Dataset3[0]
//     PlcTask Outputs/GVL.safetyOut[21] <-> Out/Out_Dataset3[1]
//     PlcTask Outputs/GVL.safetyOut[22] <-> Out/Out_Dataset3[2]
//     PlcTask Outputs/GVL.safetyOut[23] <-> Out/Out_Dataset3[3]
//     PlcTask Outputs/GVL.safetyOut[24] <-> Out/Out_Dataset3[4]
//     PlcTask Outputs/GVL.safetyOut[25] <-> Out/Out_Dataset3[5]
//     PlcTask Outputs/GVL.safetyOut[26] <-> Out/Out_Dataset3[6]
//     PlcTask Outputs/GVL.safetyOut[27] <-> Out/Out_Dataset3[7]
//     PlcTask Outputs/GVL.safetyOut[28] <-> Out/Out_Dataset3[8]
//     PlcTask Outputs/GVL.safetyOut[29] <-> Out/Out_Dataset3[9]
//     PlcTask Outputs/GVL.safetyOut[2] <-> Out/Out_Dataset1[2]
//     PlcTask Outputs/GVL.safetyOut[30] <-> Out/Out_Dataset4[0]
//     PlcTask Outputs/GVL.safetyOut[31] <-> Out/Out_Dataset4[1]
//     PlcTask Outputs/GVL.safetyOut[32] <-> Out/Out_Dataset4[2]
//     PlcTask Outputs/GVL.safetyOut[33] <-> Out/Out_Dataset4[3]
//     PlcTask Outputs/GVL.safetyOut[34] <-> Out/Out_Dataset4[4]
//     PlcTask Outputs/GVL.safetyOut[35] <-> Out/Out_Dataset4[5]
//     PlcTask Outputs/GVL.safetyOut[36] <-> Out/Out_Dataset4[6]
//     PlcTask Outputs/GVL.safetyOut[37] <-> Out/Out_Dataset4[7]
//     PlcTask Outputs/GVL.safetyOut[38] <-> Out/Out_Dataset4[8]
//     PlcTask Outputs/GVL.safetyOut[39] <-> Out/Out_Dataset4[9]
//     PlcTask Outputs/GVL.safetyOut[3] <-> Out/Out_Dataset1[3]
//     PlcTask Outputs/GVL.safetyOut[40] <-> Out/Out_Dataset5[0]
//     PlcTask Outputs/GVL.safetyOut[41] <-> Out/Out_Dataset5[1]
//     PlcTask Outputs/GVL.safetyOut[42] <-> Out/Out_Dataset5[2]
//     PlcTask Outputs/GVL.safetyOut[43] <-> Out/Out_Dataset5[3]
//     PlcTask Outputs/GVL.safetyOut[44] <-> Out/Out_Dataset5[4]
//     PlcTask Outputs/GVL.safetyOut[45] <-> Out/Out_Dataset5[5]
//     PlcTask Outputs/GVL.safetyOut[46] <-> Out/Out_Dataset5[6]
//     PlcTask Outputs/GVL.safetyOut[47] <-> Out/Out_Dataset5[7]
//     PlcTask Outputs/GVL.safetyOut[48] <-> Out/Out_Dataset5[8]
//     PlcTask Outputs/GVL.safetyOut[49] <-> Out/Out_Dataset5[9]
//     PlcTask Outputs/GVL.safetyOut[4] <-> Out/Out_Dataset1[4]
//     PlcTask Outputs/GVL.safetyOut[5] <-> Out/Out_Dataset1[5]
//     PlcTask Outputs/GVL.safetyOut[6] <-> Out/Out_Dataset1[6]
//     PlcTask Outputs/GVL.safetyOut[7] <-> Out/Out_Dataset1[7]
//     PlcTask Outputs/GVL.safetyOut[8] <-> Out/Out_Dataset1[8]
//     PlcTask Outputs/GVL.safetyOut[9] <-> Out/Out_Dataset1[9]
//   kittingDeca/kittingDeca Instance <-> NC-Task 1 SAF/Axes/fr0
//     PlcTask Inputs/GVL.fr[0].AxisRef.NcToPlc <-> Outputs/ToPlc
//     PlcTask Inputs/GVL.fr_actTorque[0] <-> Outputs/ToPlc/ActTorque
//     PlcTask Outputs/GVL.fr[0].AxisRef.PlcToNc <-> Inputs/FromPlc
//   kittingDeca/kittingDeca Instance <-> NC-Task 1 SAF/Axes/fr1
//     PlcTask Inputs/GVL.fr[1].AxisRef.NcToPlc <-> Outputs/ToPlc
//     PlcTask Inputs/GVL.fr_actTorque[1] <-> Outputs/ToPlc/ActTorque
//     PlcTask Outputs/GVL.fr[1].AxisRef.PlcToNc <-> Inputs/FromPlc
//   kittingDeca/kittingDeca Instance <-> NC-Task 1 SAF/Axes/lc0
//     PlcTask Inputs/GVL.lc[0].lateral.AxisRef.NcToPlc <-> Outputs/ToPlc
//     PlcTask Outputs/GVL.lc[0].lateral.AxisRef.PlcToNc <-> Inputs/FromPlc
//   kittingDeca/kittingDeca Instance <-> NC-Task 1 SAF/Axes/lc1
//     PlcTask Inputs/GVL.lc[1].lateral.AxisRef.NcToPlc <-> Outputs/ToPlc
//     PlcTask Outputs/GVL.lc[1].lateral.AxisRef.PlcToNc <-> Inputs/FromPlc
//   kittingDeca/kittingDeca Instance <-> NC-Task 1 SAF/Axes/pm0_buf0
//     PlcTask Inputs/GVL.pm[0].buffer[0].AxisRef.NcToPlc <-> Outputs/ToPlc
//     PlcTask Outputs/GVL.pm[0].buffer[0].AxisRef.PlcToNc <-> Inputs/FromPlc
//   kittingDeca/kittingDeca Instance <-> NC-Task 1 SAF/Axes/pm0_buf1
//     PlcTask Inputs/GVL.pm[0].buffer[1].AxisRef.NcToPlc <-> Outputs/ToPlc
//     PlcTask Outputs/GVL.pm[0].buffer[1].AxisRef.PlcToNc <-> Inputs/FromPlc
//   kittingDeca/kittingDeca Instance <-> NC-Task 1 SAF/Axes/pm1_buf0
//     PlcTask Inputs/GVL.pm[1].buffer[0].AxisRef.NcToPlc <-> Outputs/ToPlc
//     PlcTask Outputs/GVL.pm[1].buffer[0].AxisRef.PlcToNc <-> Inputs/FromPlc
//   kittingDeca/kittingDeca Instance <-> NC-Task 1 SAF/Axes/pm1_buf1
//     PlcTask Inputs/GVL.pm[1].buffer[1].AxisRef.NcToPlc <-> Outputs/ToPlc
//     PlcTask Outputs/GVL.pm[1].buffer[1].AxisRef.PlcToNc <-> Inputs/FromPlc
//   kittingDeca/kittingDeca Instance <-> NC-Task 1 SAF/Axes/pm2_buf0
//     PlcTask Inputs/GVL.pm[2].buffer[0].AxisRef.NcToPlc <-> Outputs/ToPlc
//     PlcTask Outputs/GVL.pm[2].buffer[0].AxisRef.PlcToNc <-> Inputs/FromPlc
//   kittingDeca/kittingDeca Instance <-> NC-Task 1 SAF/Axes/pm2_buf1
//     PlcTask Inputs/GVL.pm[2].buffer[1].AxisRef.NcToPlc <-> Outputs/ToPlc
//     PlcTask Outputs/GVL.pm[2].buffer[1].AxisRef.PlcToNc <-> Inputs/FromPlc
//   kittingDeca/kittingDeca Instance <-> NC-Task 1 SAF/Axes/pm3_buf0
//     PlcTask Inputs/GVL.pm[3].buffer[0].AxisRef.NcToPlc <-> Outputs/ToPlc
//     PlcTask Outputs/GVL.pm[3].buffer[0].AxisRef.PlcToNc <-> Inputs/FromPlc
//   kittingDeca/kittingDeca Instance <-> NC-Task 1 SAF/Axes/pm3_buf1
//     PlcTask Inputs/GVL.pm[3].buffer[1].AxisRef.NcToPlc <-> Outputs/ToPlc
//     PlcTask Outputs/GVL.pm[3].buffer[1].AxisRef.PlcToNc <-> Inputs/FromPlc
//   kittingDeca/kittingDeca Instance <-> NC-Task 1 SAF/Axes/pm4_buf0
//     PlcTask Inputs/GVL.pm[4].buffer[0].AxisRef.NcToPlc <-> Outputs/ToPlc
//     PlcTask Outputs/GVL.pm[4].buffer[0].AxisRef.PlcToNc <-> Inputs/FromPlc
//   kittingDeca/kittingDeca Instance <-> NC-Task 1 SAF/Axes/pm4_buf1
//     PlcTask Inputs/GVL.pm[4].buffer[1].AxisRef.NcToPlc <-> Outputs/ToPlc
//     PlcTask Outputs/GVL.pm[4].buffer[1].AxisRef.PlcToNc <-> Inputs/FromPlc
//   kittingDeca/kittingDeca Instance <-> NC-Task 1 SAF/Axes/pm5_buf0
//     PlcTask Inputs/GVL.pm[5].buffer[0].AxisRef.NcToPlc <-> Outputs/ToPlc
//     PlcTask Outputs/GVL.pm[5].buffer[0].AxisRef.PlcToNc <-> Inputs/FromPlc
//   kittingDeca/kittingDeca Instance <-> NC-Task 1 SAF/Axes/pm5_buf1
//     PlcTask Inputs/GVL.pm[5].buffer[1].AxisRef.NcToPlc <-> Outputs/ToPlc
//     PlcTask Outputs/GVL.pm[5].buffer[1].AxisRef.PlcToNc <-> Inputs/FromPlc
//   kittingDeca/kittingDeca Instance <-> NC-Task 1 SAF/Axes/pm6_buf0
//     PlcTask Inputs/GVL.pm[6].buffer[0].AxisRef.NcToPlc <-> Outputs/ToPlc
//     PlcTask Outputs/GVL.pm[6].buffer[0].AxisRef.PlcToNc <-> Inputs/FromPlc
//   kittingDeca/kittingDeca Instance <-> NC-Task 1 SAF/Axes/pm6_buf1
//     PlcTask Inputs/GVL.pm[6].buffer[1].AxisRef.NcToPlc <-> Outputs/ToPlc
//     PlcTask Outputs/GVL.pm[6].buffer[1].AxisRef.PlcToNc <-> Inputs/FromPlc
//   kittingDeca/kittingDeca Instance <-> NC-Task 1 SAF/Axes/pm7_buf0
//     PlcTask Inputs/GVL.pm[7].buffer[0].AxisRef.NcToPlc <-> Outputs/ToPlc
//     PlcTask Outputs/GVL.pm[7].buffer[0].AxisRef.PlcToNc <-> Inputs/FromPlc
//   kittingDeca/kittingDeca Instance <-> NC-Task 1 SAF/Axes/pm7_buf1
//     PlcTask Inputs/GVL.pm[7].buffer[1].AxisRef.NcToPlc <-> Outputs/ToPlc
//     PlcTask Outputs/GVL.pm[7].buffer[1].AxisRef.PlcToNc <-> Inputs/FromPlc
//   kittingDeca/kittingDeca Instance <-> NC-Task 1 SAF/Axes/pm8_buf0
//     PlcTask Inputs/GVL.pm[8].buffer[0].AxisRef.NcToPlc <-> Outputs/ToPlc
//     PlcTask Outputs/GVL.pm[8].buffer[0].AxisRef.PlcToNc <-> Inputs/FromPlc
//   kittingDeca/kittingDeca Instance <-> NC-Task 1 SAF/Axes/pm8_buf1
//     PlcTask Inputs/GVL.pm[8].buffer[1].AxisRef.NcToPlc <-> Outputs/ToPlc
//     PlcTask Outputs/GVL.pm[8].buffer[1].AxisRef.PlcToNc <-> Inputs/FromPlc
//   kittingDeca/kittingDeca Instance <-> NC-Task 1 SAF/Axes/pm9_buf0
//     PlcTask Inputs/GVL.pm[9].buffer[0].AxisRef.NcToPlc <-> Outputs/ToPlc
//     PlcTask Outputs/GVL.pm[9].buffer[0].AxisRef.PlcToNc <-> Inputs/FromPlc
//   kittingDeca/kittingDeca Instance <-> NC-Task 1 SAF/Axes/pm9_buf1
//     PlcTask Inputs/GVL.pm[9].buffer[1].AxisRef.NcToPlc <-> Outputs/ToPlc
//     PlcTask Outputs/GVL.pm[9].buffer[1].AxisRef.PlcToNc <-> Inputs/FromPlc
//   kittingDeca/kittingDeca Instance <-> NC-Task 1 SAF/Axes/rem0_Lift0
//     PlcTask Inputs/GVL.rem[0].lift[0].AxisRef.NcToPlc <-> Outputs/ToPlc
//     PlcTask Outputs/GVL.rem[0].lift[0].AxisRef.PlcToNc <-> Inputs/FromPlc
//   kittingDeca/kittingDeca Instance <-> NC-Task 1 SAF/Axes/rem0_Lift1
//     PlcTask Inputs/GVL.rem[0].lift[1].AxisRef.NcToPlc <-> Outputs/ToPlc
//     PlcTask Outputs/GVL.rem[0].lift[1].AxisRef.PlcToNc <-> Inputs/FromPlc
//   kittingDeca/kittingDeca Instance <-> NC-Task 1 SAF/Axes/rem1_Lift0
//     PlcTask Inputs/GVL.rem[1].lift[0].AxisRef.NcToPlc <-> Outputs/ToPlc
//     PlcTask Outputs/GVL.rem[1].lift[0].AxisRef.PlcToNc <-> Inputs/FromPlc
//   kittingDeca/kittingDeca Instance <-> NC-Task 1 SAF/Axes/rem1_Lift1
//     PlcTask Inputs/GVL.rem[1].lift[1].AxisRef.NcToPlc <-> Outputs/ToPlc
//     PlcTask Outputs/GVL.rem[1].lift[1].AxisRef.PlcToNc <-> Inputs/FromPlc
//   kittingDeca/kittingDeca Instance <-> NC-Task 1 SAF/Axes/rem2_Lift0
//     PlcTask Inputs/GVL.rem[2].lift[0].AxisRef.NcToPlc <-> Outputs/ToPlc
//     PlcTask Outputs/GVL.rem[2].lift[0].AxisRef.PlcToNc <-> Inputs/FromPlc
//   kittingDeca/kittingDeca Instance <-> NC-Task 1 SAF/Axes/rem2_Lift1
//     PlcTask Inputs/GVL.rem[2].lift[1].AxisRef.NcToPlc <-> Outputs/ToPlc
//     PlcTask Outputs/GVL.rem[2].lift[1].AxisRef.PlcToNc <-> Inputs/FromPlc
//   kittingDeca/kittingDeca Instance <-> NC-Task 1 SAF/Axes/rem3_Lift0
//     PlcTask Inputs/GVL.rem[3].lift[0].AxisRef.NcToPlc <-> Outputs/ToPlc
//     PlcTask Outputs/GVL.rem[3].lift[0].AxisRef.PlcToNc <-> Inputs/FromPlc
//   kittingDeca/kittingDeca Instance <-> NC-Task 1 SAF/Axes/rem3_Lift1
//     PlcTask Inputs/GVL.rem[3].lift[1].AxisRef.NcToPlc <-> Outputs/ToPlc
//     PlcTask Outputs/GVL.rem[3].lift[1].AxisRef.PlcToNc <-> Inputs/FromPlc
//   kittingDeca/kittingDeca Instance <-> NC-Task 1 SAF/Axes/rem4_Lift0
//     PlcTask Inputs/GVL.rem[4].lift[0].AxisRef.NcToPlc <-> Outputs/ToPlc
//     PlcTask Outputs/GVL.rem[4].lift[0].AxisRef.PlcToNc <-> Inputs/FromPlc
//   kittingDeca/kittingDeca Instance <-> NC-Task 1 SAF/Axes/rem4_Lift1
//     PlcTask Inputs/GVL.rem[4].lift[1].AxisRef.NcToPlc <-> Outputs/ToPlc
//     PlcTask Outputs/GVL.rem[4].lift[1].AxisRef.PlcToNc <-> Inputs/FromPlc
//   kittingDeca/kittingDeca Instance <-> NC-Task 1 SAF/Axes/rem5_Lift0
//     PlcTask Inputs/GVL.rem[5].lift[0].AxisRef.NcToPlc <-> Outputs/ToPlc
//     PlcTask Outputs/GVL.rem[5].lift[0].AxisRef.PlcToNc <-> Inputs/FromPlc
//   kittingDeca/kittingDeca Instance <-> NC-Task 1 SAF/Axes/rem5_Lift1
//     PlcTask Inputs/GVL.rem[5].lift[1].AxisRef.NcToPlc <-> Outputs/ToPlc
//     PlcTask Outputs/GVL.rem[5].lift[1].AxisRef.PlcToNc <-> Inputs/FromPlc
//   kittingDeca/kittingDeca Instance <-> NC-Task 1 SAF/Axes/rem6_Lift0
//     PlcTask Inputs/GVL.rem[6].lift[0].AxisRef.NcToPlc <-> Outputs/ToPlc
//     PlcTask Outputs/GVL.rem[6].lift[0].AxisRef.PlcToNc <-> Inputs/FromPlc
//   kittingDeca/kittingDeca Instance <-> NC-Task 1 SAF/Axes/rem6_Lift1
//     PlcTask Inputs/GVL.rem[6].lift[1].AxisRef.NcToPlc <-> Outputs/ToPlc
//     PlcTask Outputs/GVL.rem[6].lift[1].AxisRef.PlcToNc <-> Inputs/FromPlc
//   kittingDeca/kittingDeca Instance <-> NC-Task 1 SAF/Axes/rem7_Lift0
//     PlcTask Inputs/GVL.rem[7].lift[0].AxisRef.NcToPlc <-> Outputs/ToPlc
//     PlcTask Outputs/GVL.rem[7].lift[0].AxisRef.PlcToNc <-> Inputs/FromPlc
//   kittingDeca/kittingDeca Instance <-> NC-Task 1 SAF/Axes/rem7_Lift1
//     PlcTask Inputs/GVL.rem[7].lift[1].AxisRef.NcToPlc <-> Outputs/ToPlc
//     PlcTask Outputs/GVL.rem[7].lift[1].AxisRef.PlcToNc <-> Inputs/FromPlc
//   kittingDeca/kittingDeca Instance <-> NC-Task 1 SAF/Axes/rem8_Lift0
//     PlcTask Inputs/GVL.rem[8].lift[0].AxisRef.NcToPlc <-> Outputs/ToPlc
//     PlcTask Outputs/GVL.rem[8].lift[0].AxisRef.PlcToNc <-> Inputs/FromPlc
//   kittingDeca/kittingDeca Instance <-> NC-Task 1 SAF/Axes/rem8_Lift1
//     PlcTask Inputs/GVL.rem[8].lift[1].AxisRef.NcToPlc <-> Outputs/ToPlc
//     PlcTask Outputs/GVL.rem[8].lift[1].AxisRef.PlcToNc <-> Inputs/FromPlc
//   kittingDeca/kittingDeca Instance <-> NC-Task 1 SAF/Axes/rem9_Lift0
//     PlcTask Inputs/GVL.rem[9].lift[0].AxisRef.NcToPlc <-> Outputs/ToPlc
//     PlcTask Outputs/GVL.rem[9].lift[0].AxisRef.PlcToNc <-> Inputs/FromPlc
//   kittingDeca/kittingDeca Instance <-> NC-Task 1 SAF/Axes/rem9_Lift1
//     PlcTask Inputs/GVL.rem[9].lift[1].AxisRef.NcToPlc <-> Outputs/ToPlc
//     PlcTask Outputs/GVL.rem[9].lift[1].AxisRef.PlcToNc <-> Inputs/FromPlc

CONFIGURATION kittingDeca
    RESOURCE PLC ON TwinCAT3
        TASK PlcTask(INTERVAL := T#2ms, PRIORITY := 12);
        TASK VISU_TASK(INTERVAL := T#200000us, PRIORITY := 16);
        PROGRAM MAIN WITH PlcTask : MAIN;
        PROGRAM VisuElems_Visu_Prg WITH VISU_TASK : VisuElems.Visu_Prg;
    END_RESOURCE
END_CONFIGURATION

// ---- GVLs/kitting deca/axis/ST_MotionAxis_MC.TcDUT
TYPE ST_MotionAxis_MC :
STRUCT
	rVelocity						: 	LREAL   						;
	rVelocity2						: 	LREAL   						;
	rMaxVelocity					:	LREAL							;	
	rAcceleration					:	LREAL							;
	rMaxAcceleration				:	LREAL							;
	rDeceleration					:	LREAL   						;
	rMaxDeceleration				:	LREAL							;
	rJerk							:	LREAL							;
	rMaxJerk						:	LREAL							;
	rPosition						:	LREAL							;
	rSetPosDistance					:	LREAL							;
	rSetPos							: 	LREAL							;	
	rDistance						:   LREAL							;
	rDistance2						:   LREAL							;	
	
	rActualPosSet					:	LREAL							;//ADD BY EVAN 
	rVelocitySet					: 	LREAL   						;//ADD BY EVAN 	
	xHoming							:	BOOL							;//ADD BY EVAN 
	
	rMaxDistance					:	LREAL							;
	bLimit							:   BOOL							;
	bNegLim							:   BOOL							;
	bPosLim							:	BOOL							;
	bNegSen							:   BOOL							;
	bPosSen							:	BOOL							;
	bPositionSensor					:	BOOL							;
	rHomePos						:	LREAL							;
	rActualPos						:	LREAL							;
	PosDiff							:	LREAL							;
	rActualCurr						:	LREAL							;
	axisDirection					:	MC_Direction					;
	
	rVeloPers						: 	LREAL							;
	rAccPers						: 	LREAL							;   
	rDecPers						: 	LREAL							;                                             					
	SetHomePos						: 	LREAL							;
	HomeVelo						: 	LREAL							;
	PosDiffTarget					: 	LREAL							;
	rFirstpos						: 	LREAL							;
	iAxisID							:	INT								;
	xhsHomingStart					: 	BOOL							;
	xHomingDone						: 	BOOL							;
	xForceControlStart				: 	BOOL							;
	xFoceControlDone				:	BOOL							;	
	xMoveABSDone					: 	BOOL							;
	xMoveRelDone					:	BOOL							;
	bInCouple						:	BOOL							;//Flag Axis is coupled 
    xMuteAxisErrorMessages			:	BOOL							;                                         					
	//Visible/Hide HMI interfaces                   					
	bHomeButtonShow					:	BOOL							; 
	bNegSensorShow					:	BOOL							; 
	bPosSensorShow					:	BOOL							;
	bBacklashShow					:	BOOL							;
	bUnitDegShow					:	BOOL							;
    bJerkShow						:	BOOL							; 
	bStopButtonShow					:	BOOL							; 
	   
	
	bMoveAbsHMI						:	BOOL;
	rVelocityHMI 					: 	LREAL;
	rActualPosHMI					:	LREAL							;//ADD BY EVAN
	bMChomingEnable					:	BOOL							;                                         				
	// backlash compensation                        	
	rBacklashvalue					:	LREAL							;
	xbacklashEnable					:	BOOL							;                        		                					
	bdirFW							:	BOOL							;// on hard stop homing , define the direction of rotation
	
	ModOp					 		: 	SINT							;// Axis operation mode (8 )

//	==============================	Beckhoff Tc2_MC2 library(motion)	==================================
	mcPower 						: 	MC_Power					    ;(*	Axis power, enable/disable																			*)
	mcAxisStates					:	MC_AxisStates					;(*	Driver Feedback, curr motor stage 																	*)
	mcHalt							: 	MC_Halt							;(*	Stops an axis with a defined braking ramp															*)
	mcHome							: 	MC_Home							;(*	Axis homing scenario and execution																	*)
	mcJog							: 	MC_Jog							;(*	Axis Joging BW/FW																					*)	
	mcMoveAbsolute					: 	MC_MoveAbsolute					;(*	Axis GoTo Absolute position																			*)	
	mcMoveRelative					: 	MC_MoveRelative					;(*	Axis GoTo Step by SetPos +/- actual position														*)
	mcMoveVelocity					: 	MC_MoveVelocity					;(*	Axis GoTo with constant velocity														*)
	mcReadStatus					: 	MC_ReadStatus					;(*	Read Axis statuses from driver																		*)
	mcReset							: 	MC_Reset						;(*	Reset Driver																						*)
	mcStop							: 	MC_Stop							;(*	Stop Driver																							*)
	mcReadActualPosition			:	MC_ReadActualPosition			;(*	Read the current axis position																		*)
	mcSetpoint						: 	MC_SetPosition					;(*	Sets the current axis position to a parameterizable value											*)
	mcWriteBoolParameter			: 	MC_WriteBoolParameter			;(*	Write bool param to driver																			*)
	mcReadBoolParameter				:	MC_ReadBoolParameter			;(*	Read bool param from driver																			*)
	mcAxisParameter					:   MC_AxisParameter				;(*	Data type is used in conjunction with function blocks for reading and writing of axis parameters	*)
	CoeWrt							:	FB_EcCoESdoWrite;									
	
//	======================================================================================================	

//
	iSdoWrite	:INT; //6:clear encoder
	sNetID : STRING;
	nSlaveAddr	:UINT;
	nSubIndex	: BYTE;
	nIndex	: WORD;
	
	iCoeWrt	: INT;
	rToqueLimitSet	: LREAL	:= 350;
	rActTorque	: LREAL;
	xTorqueErr	: BOOL;
END_STRUCT
END_TYPE

// ---- GVLs/kitting deca/E_CMD_ConverterMotor.TcDUT
{attribute 'qualified_only'}
{attribute 'strict'}
TYPE E_CMD_ConverterMotor :
(
	STOP	:=0,
	FORWARD	:=1,
	BACKWARE	:=2,
	JOG_POS	:=3,
	JOG_NEG	:=4,
	FREE_STOP	:=5,
	SLOWDOWN_STOP	:=6,
	RESET	:= 7
);
END_TYPE

// ---- GVLs/kitting deca/fixture rotation/fixtureRotation_Module.TcDUT
TYPE fixtureRotation_Module :
STRUCT
	power_axis	: BOOL;
	contactor_axis : BOOL;	
	mcAxis 					: FB_MotionAxis_MC;
	st_mcAxis 				: ST_MotionAxis_MC;
	AxisRef					: AXIS_REF;
	valve	:Valve;
	limit_sensor : ARRAY[0..2]OF BOOL;
END_STRUCT
END_TYPE

// ---- GVLs/kitting deca/lateral conveyor/BeltOut.TcDUT
TYPE BeltOut :
STRUCT
	belt : Belt;
	photo_sensor :ARRAY[0..2]OF BOOL;
END_STRUCT
END_TYPE

// ---- GVLs/kitting deca/lateral conveyor/Lateral.TcDUT
TYPE Lateral :
STRUCT
	
	power_axis	: BOOL;
	contactor_axis : BOOL;	
	mcAxis 					: FB_MotionAxis_MC;
	st_mcAxis 				: ST_MotionAxis_MC;
	AxisRef					: AXIS_REF;
	valve_lift	:Valve;
	valve_clamp	:	ARRAY[0..1]OF Valve;
	limit_sensor : ARRAY[0..2]OF BOOL;
	

END_STRUCT
END_TYPE

// ---- GVLs/kitting deca/lateral conveyor/LateralBuf_Module.TcDUT
TYPE LateralBuf_Module :
STRUCT

	power_beltConv		: BOOL;
	contactor_beltConv	: BOOL;	

	belt	: ARRAY[0..2] OF Belt;
	photo_sensor :ARRAY[0..2]OF BOOL;
	valve_stopper : ARRAY [0..5] OF Valve;
	
	
END_STRUCT
END_TYPE

// ---- GVLs/kitting deca/lateral conveyor/Roller_LC.TcDUT
TYPE Roller_LC :
STRUCT
	roller : Roller;	
	photo_sensor :BOOL;
END_STRUCT
END_TYPE

// ---- GVLs/kitting deca/lateral conveyor/LateralRecy_Module.TcDUT
TYPE LateralRecy_Module :
STRUCT
	pressure_sensor	: BOOL;
	power_beltConv		: BOOL;
	contactor_beltConv	: BOOL;	
	rollerIn : Roller_LC;
	rollerOut : Roller_LC;
	belt_out : BeltOut;
	lateral	: Lateral;
	valve_stopper : ARRAY [0..1] OF Valve;
	valve_guide : ARRAY [0..1] OF Valve;
END_STRUCT
END_TYPE

// ---- GVLs/kitting deca/picking module/Belt.TcDUT
TYPE Belt :
STRUCT
	//cmd  AT%Q*	: UINT;
	//freq AT%Q*	: UINT;
	fbconverter	: FB_Converter;
END_STRUCT
END_TYPE

// ---- GVLs/kitting deca/picking module/Inner_conveyor.TcDUT
TYPE Inner_conveyor :
STRUCT
	belt	: ARRAY[0..2] OF Belt;
	valve	: ARRAY[0..2] OF Valve;
	rfid	: ARRAY[0..1] OF RFID;
	photo_sensor	: ARRAY[0..5] OF BOOL;
END_STRUCT
END_TYPE

// ---- GVLs/kitting deca/ST_Converter.TcDUT
TYPE ST_Converter :
STRUCT
	
	
	sNetID : STRING;
	nSlaveAddr	:UINT;
	nSubIndex	:ARRAY [0..13] OF BYTE;
	nIndex	:ARRAY [0..13] OF WORD;
	iSdoWrite	:ARRAY [0..13] OF INT; 
	
	iCoeWrt	: INT;
END_STRUCT
END_TYPE

// ---- GVLs/kitting deca/ST_heightDetection.TcDUT
TYPE ST_heightDetection :
STRUCT
		
	sNetID : STRING;
	nSlaveAddr	: UINT;
	nSubIndex	: BYTE;
	nIndex	: WORD;
	iSdoWrite	: DWORD; 
	iSdoRead	: DWORD; 
END_STRUCT
END_TYPE

// ---- POUs/bagmachines/AdsArr.TcDUT
TYPE AdsArr :
STRUCT
	inArr	: ARRAY[0..31] OF WORD;
	outArr	: ARRAY[0..31] OF WORD;
END_STRUCT
END_TYPE

// ---- POUs/bagmachines/BagCmd.TcDUT
{attribute 'qualified_only'}
{attribute 'strict'}
TYPE BagCmd:
(
	DO_NOTHING := 0,
    INSERT_BAG_HOLDER := 1,
    REMOVE_BAG_HOLDER := 2,
	STOP	:=3
);
END_TYPE

// ---- POUs/bagmachines/BagDetectionCmd.TcDUT
{attribute 'qualified_only'}
{attribute 'strict'}
TYPE BagDetectionCmd:
(
	DO_NOTHING := 0,
    GET_RESULT_FROM_CAMERA := 1,
    RESET_CAMERA := 2
);
END_TYPE

// ---- POUs/bagmachines/BagDetectionStatus.TcDUT
{attribute 'qualified_only'}
{attribute 'strict'}
TYPE BagDetectionStatus:
(
    UNKNOWN := 0,
    OKAY := 1,
    NG := 2,
	ERROR := 3
);
END_TYPE

// ---- POUs/bagmachines/BagHeightStatus.TcDUT
{attribute 'qualified_only'}
{attribute 'strict'}
TYPE BagHeightStatus:
(
    UNKNOWN := 0,
    OKAY := 1,
    NG := 2,
	ERROR := 3
);
END_TYPE

// ---- POUs/bagmachines/BagHolderStatus.TcDUT
{attribute 'qualified_only'}
{attribute 'strict'}
TYPE BagHolderStatus:
(
	UNKNOWN	:=0,
    DOWN := 1,
    UP := 2
);
END_TYPE

// ---- POUs/bagmachines/BagMachineStatus.TcDUT
{attribute 'qualified_only'}
{attribute 'strict'}
TYPE BagMachineStatus:
(
    OFF := 0,
    BUSY := 1,
    READY := 2,
	RESET	:=3,
    ERROR := 4,
	STOPPED := 5
);
END_TYPE

// ---- POUs/bagmachines/BagStatus.TcDUT
{attribute 'qualified_only'}
{attribute 'strict'}
TYPE BagStatus:
(
	UNKNOWN :=0,
    READY := 1,
    INSERTED := 2,
    REMOVED := 3
    //CAMERA_OK := 3,
    //CAMERA_ERROR := 4
);
END_TYPE

// ---- POUs/bagmachines/E_HeightDetection.TcDUT
{attribute 'qualified_only'}
{attribute 'strict'}
TYPE E_HeightDetection :
(
	DO_NOTHING := 0,
	SET_PROGRAM	:= 1,
	READ_HEIGHT	:= 2
);
END_TYPE

// ---- POUs/G_HMI.TcGVL
{attribute 'qualified_only'}
VAR_GLOBAL
	iMainFrame : INT;
	iReM: INT;
	iPM	: INT;
	iOthers	: INT;
	iLc	: INT;
	iLb	: INT;
	iFr	: INT;
END_VAR

// ---- POUs/GVL.TcGVL
{attribute 'qualified_only'}
VAR_GLOBAL CONSTANT
	netId_bagmachie :ARRAY[0..2] OF STRING	:=['192.168.11.160.1.1','192.168.11.161.1.1','192.168.11.162.1.1'];//[0]:bag_opener;[1]:bag_closer;[2]:bag_compactor
END_VAR
VAR_GLOBAL

	
	
	rem : ARRAY[0..9] OF Replenishment_Module;
	pm	: ARRAY[0..9] OF Picking_Module;
	pmOthers	:ARRAY[0..4] OF PM_others;
	lc	: ARRAY[0..1] OF LateralRecy_Module;
	lb	: ARRAY[0..1] OF LateralBuf_Module;
	fr	: ARRAY[0..1] OF fixtureRotation_Module;
	
	
    stByte : REFERENCE TO ST_byte;
	ibyteNum			:ARRAY[1..32] OF  INT ;
	stMeasuringLC : ST_byte;
	byteLC AT%I*:ARRAY [1..32] OF BYTE;
	rfidIn AT%I*:ARRAY [0..31] OF BYTE;
	rfidOut AT%Q*:ARRAY [0..31] OF BYTE;
	arIn	: ARRAY[0..3] OF ST_IO_byte;
	arOut	: ARRAY[0..3] OF ST_IO_byte;
	n: INT;
	
	fb_remIOmapping	: ARRAY[0..9] OF FB_remIOmapping;
	fb_remAxisMapping	: ARRAY[0..19] OF FB_remAxisMapping;
	stAxisCtrl_Lift	: ARRAY[0..19]OF ST_axisCtrl;
	fbAxisCtrl_Lift	: ARRAY [0..19] OF FB_axisCtrl;
	
	

	fb_rmIOmapping	: ARRAY[0..4] OF FB_rmIOmapping;
	fb_pmAxisMapping	: ARRAY[0..19] OF FB_pmAxisMapping;
	stAxisCtrl_Buffer	: ARRAY[0..19]OF ST_axisCtrl;
	fbAxisCtrl_Buffer	: ARRAY [0..19] OF FB_axisCtrl;
	
	fbconverter	:ARRAY [0..13] OF  FB_Converter;
	stConverter	:ARRAY [0..13] OF  ST_Converter;
	
	ref_fbconverterMotor	:   ARRAY[0..57] OF POINTER TO FB_Converter;	
	

	
	fb_lcIOmappiing : ARRAY [0..1] OF FB_lcIOmapping;
	//fb_lcAxis	: ARRAY[0..1] OF FB_MotionAxis_MC;
	//stAxis_LC	: ARRAY[0..1] OF ST_MotionAxis_MC;
	stAxisCtrl_LC	: ARRAY[0..1]OF ST_axisCtrl;
	fbAxisCtrl_LC	: ARRAY [0..1] OF FB_axisCtrl;
	
	fb_lbIOmappiing : ARRAY [0..1] OF FB_lbIOmapping;
	
	
	
	fb_frIOmappiing : ARRAY [0..1] OF FB_frIOmapping;
	//fb_frAxis	: ARRAY[0..1] OF FB_MotionAxis_MC;
	//stAxis_FR	: ARRAY[0..1] OF ST_MotionAxis_MC;	
	stAxisCtrl_FR	: ARRAY[0..1]OF ST_axisCtrl;
	fbAxisCtrl_FR	: ARRAY [0..1] OF FB_axisCtrl;	
	
	
	safetyin AT%I*	: ARRAY[0..49]OF BYTE;
	safetyOut AT%Q*	: ARRAY[0..49]OF BYTE;
	
	

	adsArr_bagMachine	: ARRAY[0..2] OF AdsArr;
	adsread		: ARRAY[0..2] OF ADSREAD;
	adswrite	: ARRAY[0..2] OF ADSWRITE;
	bread		: ARRAY[0..2] OF BOOL;
	bwrite		: ARRAY[0..2] OF BOOL;
	
	fb_bagOpener	: FB_BagOpener;
	fb_bagCloser	: FB_BagCloser;
	fb_bagCompactor	: FB_BagCompactor;
	
	adsReadByName	: FB_ReadAdsSymByName;
	adsReadEvents	: FB_AdsReadEvents;
	
	bBagmachine_test	: BOOL;
	
	fr_actTorque	AT%I*	: ARRAY[0..1]OF LREAL ;
	fr_torqueLimitSet		: ARRAY[0..1]OF LREAL :=[120,120] ;
	
	arrValve_PM	: ARRAY[0..99]OF FB_valve;
	arrValve_Rem	: ARRAY[0..119] OF FB_valve;
	
	fb_heightDetection	: FB_heightDetection;
	stHeightDetection	: ST_heightDetection;
END_VAR

// ---- POUs/G_IO.TcGVL
{attribute 'global_init_slot' := '40600'}
VAR_GLOBAL CONSTANT
	{attribute 'global_init_slot'}
	DiMouduleMAX 			:	INT	:=	100;
	{attribute 'global_init_slot'}
	DOMODULEMAX 			:	INT	:=	100;
END_VAR

VAR_GLOBAL
	{attribute 'TcContextName':='PlcTask1'}
	arDI	AT%I*		: ARRAY[0..DiMouduleMAX ] OF ST_IO_16;		//  links to Digital input  Modules 
	{attribute 'TcContextName':='PlcTask1'}
	arDO	AT%Q*		: ARRAY[0..DOMODULEMAX ] OF ST_IO_16;		//  links to Digital output Modules

	iDiMouduleMAX		: INT := 100 							; 		//Number of DI module 
	iDOModuleMax		: INT := 100 							; 		//Number of DO module 


	stDIO				: ST_DIO 							;		// struct DIO for use in plc program
		
	{attribute 'TcContextName':='PlcTask1'}
   	
	
END_VAR

// ---- POUs/MAIN.TcPOU
PROGRAM MAIN
VAR
	test_bool:BOOL;
	test_int:INT;
	test_real:REAL;
	test_string:STRING;
	test_arr_int:ARRAY[1..10] OF INT;
	test_word:WORD;
	test_arr_bool:ARRAY[1..3] OF BOOL;
	test_structure:user_defined_structure;
	test_arr_string:ARRAY[1..3] OF STRING;
	
	fb_Time : FB_LocalSystemTime;

	byte1 : BYTE;
	string1 :STRING;

	iInit	: int;
	i	: INT;
	j	: INT;
	
	ton_1ms	: TON;
	iAds: INT;
	
	xErr_converterMotors	: BOOL;
	xErr_servoMoters	: BOOL;
	xError	: BOOL;

	xReset	: BOOL;
	
	

	iReset: INT;
	
END_VAR

fb_Time(bEnable := TRUE); 

M_mappingIO();
M_measuringLC();
M_rfid();
runEveryCycle();
M_ReM();
//M_ads_bagmachines();
safetyConfig();
agingTestConfig();



CASE iInit OF
	0:
		FOR i:=0 TO 57 DO
			GVL.ref_fbconverterMotor[i]^.bSetParaEx	:= FALSE;
		END_FOR
		FOR i:=0 TO 99 DO
			GVL.arrValve_PM[i].bStart	:= FALSE;
			GVL.arrValve_PM[i].bStop	:= FALSE;
		END_FOR			
	1://set parameters for all converter motors
		FOR i:=0 TO 57 DO
			GVL.ref_fbconverterMotor[i]^.bSetParaEx	:= TRUE;
		END_FOR
		IF GVL.ref_fbconverterMotor[57]^.xDone THEN
			iInit	:=2;
		END_IF
	2://set parameters for all converter motors
		FOR i:=0 TO 57 DO
			GVL.ref_fbconverterMotor[i]^.bSetParaEx	:= FALSE;
		END_FOR
		iInit	:=0;
	3://run all converter motors
		FOR i:=0 TO 57 DO
			GVL.ref_fbconverterMotor[i]^.cmd	:=INT_TO_UINT(E_CMD_ConverterMotor.BACKWARE);
			GVL.ref_fbconverterMotor[i]^.freq	:= 2000;
		END_FOR
	4://stop all converter moters
		FOR i:=0 TO 57 DO
			GVL.ref_fbconverterMotor[i]^.cmd	:= 0;
			GVL.ref_fbconverterMotor[i]^.freq	:= 0;
		END_FOR
		iInit	:=0;
	5://all lift axis servo on
		FOR i:=0 TO 19 DO
			GVL.stAxisCtrl_Lift[i].iCmd	:= 1;
			GVL.stAxisCtrl_Buffer[i].iCmd	:= 1;
		END_FOR
		FOR i:=0 TO 1 DO
			GVL.stAxisCtrl_LC[i].iCmd	:= 1;
			GVL.stAxisCtrl_FR[i].iCmd	:= 1;
		END_FOR
		iInit	:=0;
	6://all lift axis run
		FOR i:=0 TO 19 DO
			GVL.stAxisCtrl_Lift[i].rPosition	:= 0;
			GVL.stAxisCtrl_Lift[i].iSpeed	:= 200;
			GVL.stAxisCtrl_Lift[i].iCmd	:= 10;
		END_FOR
		iInit	:=0;
	7://all buffer axis run
		FOR i:=0 TO 19 DO
			GVL.stAxisCtrl_Buffer[i].rPosition	:= 250;
			GVL.stAxisCtrl_Buffer[i].iSpeed	:= 100;
			GVL.stAxisCtrl_Buffer[i].iCmd	:= 20;
		END_FOR	
		iInit	:=0;
	8://all lift axis stop
		FOR i:=0 TO 19 DO
			GVL.stAxisCtrl_Lift[i].iCmd	:= 100;
			GVL.stAxisCtrl_Buffer[i].iCmd	:= 100;
		END_FOR	
		FOR i:=0 TO 1 DO
			GVL.stAxisCtrl_LC[i].iCmd	:= 100;
			GVL.stAxisCtrl_FR[i].iCmd	:= 100;
		END_FOR		
		FOR i:=0 TO 57 DO
			GVL.ref_fbconverterMotor[i]^.cmd	:= 0;
			GVL.ref_fbconverterMotor[i]^.freq	:= 0;
		END_FOR
		FOR i:=0 TO 99 DO
			GVL.arrValve_PM[i].bStop	:= TRUE;
		END_FOR	
		FOR i:=0 TO 119 DO
			GVL.arrValve_Rem[i].bStop	:= TRUE;
		END_FOR			
		iInit	:=0;		
	9://check error
		IF M_checkError() THEN
			iInit	:=0;
		END_IF
	
	10://reset error
		IF M_reset() THEN
			iInit	:=0;
		END_IF		
	11://
		FOR i:=0 TO 1 DO
			GVL.stAxisCtrl_LC[i].rPosition	:= -800;
			GVL.stAxisCtrl_LC[i].iSpeed	:= 600;
			GVL.stAxisCtrl_LC[i].iCmd	:= 10;
		END_FOR
		iInit	:=0;	
	12://
		FOR i:=0 TO 1 DO
			GVL.stAxisCtrl_FR[i].rPosition	:= -170;
			GVL.stAxisCtrl_FR[i].iSpeed	:= 200;
			GVL.stAxisCtrl_FR[i].iCmd	:= 10;
		END_FOR
		iInit	:=0;	
	13://aging test valve of pm
		FOR i:=0 TO 99 DO
			GVL.arrValve_PM[i].bStart	:= TRUE;
		END_FOR
		iInit	:=0;
	14://aging test valve of rem
		FOR i:=0 TO 119 DO
			GVL.arrValve_Rem[i].bStart	:= TRUE;
		END_FOR		
		iInit	:=0;	

END_CASE

GVL.fb_bagOpener(ams_net_id:=GVL.netId_bagmachie[0]);
GVL.fb_bagCloser(ams_net_id:=GVL.netId_bagmachie[1]);
GVL.fb_bagCompactor(ams_net_id:=GVL.netId_bagmachie[2]);
IF test_bool THEN
	ADSLOGSTR(msgCtrlMask:= ADSLOG_MSGTYPE_LOG,msgFmtStr:='msg:log',strArg:='MSG ARG');
	test_bool	:= FALSE;
END_IF
GVL.stHeightDetection.sNetID:='192.168.11.159.9.1';
GVL.stHeightDetection.nSlaveAddr:=1001;
GVL.fb_heightDetection(stHeightDetection:=GVL.stHeightDetection);

ACTION agingTestConfig:
GVL.stConverter[0].sNetID	:= '192.168.11.159.5.1';
GVL.stConverter[0].nSlaveAddr	:= 1003;//lb[0]
GVL.stConverter[1].sNetID	:= '192.168.11.159.5.1';
GVL.stConverter[1].nSlaveAddr	:= 1005;//lc[0]
GVL.stConverter[2].sNetID	:= '192.168.11.159.5.1';
GVL.stConverter[2].nSlaveAddr	:= 1008;//pm[0]_inner
GVL.stConverter[3].sNetID	:= '192.168.11.159.5.1';
GVL.stConverter[3].nSlaveAddr	:= 1009;//pm[0]_outer
GVL.stConverter[4].sNetID	:= '192.168.11.159.5.1';
GVL.stConverter[4].nSlaveAddr	:= 1018;//pm[1]_inner
GVL.stConverter[5].sNetID	:= '192.168.11.159.5.1';
GVL.stConverter[5].nSlaveAddr	:= 1019;//pm[1]_outer
GVL.stConverter[6].sNetID	:= '192.168.11.159.5.1';
GVL.stConverter[6].nSlaveAddr	:= 1026;//pm[2]_inner
GVL.stConverter[7].sNetID	:= '192.168.11.159.5.1';
GVL.stConverter[7].nSlaveAddr	:= 1027;//pm[2]_outer
GVL.stConverter[8].sNetID	:= '192.168.11.159.5.1';
GVL.stConverter[8].nSlaveAddr	:= 1034;//pm[3]_inner
GVL.stConverter[9].sNetID	:= '192.168.11.159.5.1';
GVL.stConverter[9].nSlaveAddr	:= 1035;//pm[3]_outer
GVL.stConverter[10].sNetID	:= '192.168.11.159.5.1';
GVL.stConverter[10].nSlaveAddr	:= 1044;//pm[4]_inner
GVL.stConverter[11].sNetID	:= '192.168.11.159.5.1';
GVL.stConverter[11].nSlaveAddr	:= 1045;//pm[4]_outer
GVL.stConverter[12].sNetID	:= '192.168.11.159.5.1';
GVL.stConverter[12].nSlaveAddr	:= 1052;//lb[1]
GVL.stConverter[13].sNetID	:= '192.168.11.159.5.1';
GVL.stConverter[13].nSlaveAddr	:= 1054;//lc[1]
GVL.lb[0].belt[0].fbconverter(stConverter:=GVL.stConverter[0],iMotor:=0);
GVL.lb[0].belt[1].fbconverter(stConverter:=GVL.stConverter[0],iMotor:=1);
GVL.lb[0].belt[2].fbconverter(stConverter:=GVL.stConverter[0],iMotor:=2);
GVL.lc[0].belt_out.belt.fbconverter(stConverter:=GVL.stConverter[1],iMotor:=0);
GVL.pm[0].inConv.belt[0].fbconverter(stConverter:= GVL.stConverter[2],iMotor:=0);
GVL.pm[0].inConv.belt[1].fbconverter(stConverter:= GVL.stConverter[2],iMotor:=1);
GVL.pm[0].inConv.belt[2].fbconverter(stConverter:= GVL.stConverter[2],iMotor:=2);
GVL.pm[1].inConv.belt[0].fbconverter(stConverter:= GVL.stConverter[2],iMotor:=3);
GVL.pm[1].inConv.belt[1].fbconverter(stConverter:= GVL.stConverter[2],iMotor:=4);
GVL.pm[1].inConv.belt[2].fbconverter(stConverter:= GVL.stConverter[2],iMotor:=5);
GVL.pm[0].outConv.belt[0].fbconverter(stConverter:= GVL.stConverter[3],iMotor:=0);
GVL.pm[0].outConv.belt[1].fbconverter(stConverter:= GVL.stConverter[3],iMotor:=1);
GVL.pm[1].outConv.belt[0].fbconverter(stConverter:= GVL.stConverter[3],iMotor:=2);
GVL.pm[1].outConv.belt[1].fbconverter(stConverter:= GVL.stConverter[3],iMotor:=3);
GVL.pm[2].inConv.belt[0].fbconverter(stConverter:= GVL.stConverter[4],iMotor:=0);
GVL.pm[2].inConv.belt[1].fbconverter(stConverter:= GVL.stConverter[4],iMotor:=1);
GVL.pm[2].inConv.belt[2].fbconverter(stConverter:= GVL.stConverter[4],iMotor:=2);
GVL.pm[3].inConv.belt[0].fbconverter(stConverter:= GVL.stConverter[4],iMotor:=3);
GVL.pm[3].inConv.belt[1].fbconverter(stConverter:= GVL.stConverter[4],iMotor:=4);
GVL.pm[3].inConv.belt[2].fbconverter(stConverter:= GVL.stConverter[4],iMotor:=5);
GVL.pm[2].outConv.belt[0].fbconverter(stConverter:= GVL.stConverter[5],iMotor:=0);
GVL.pm[2].outConv.belt[1].fbconverter(stConverter:= GVL.stConverter[5],iMotor:=1);
GVL.pm[3].outConv.belt[0].fbconverter(stConverter:= GVL.stConverter[5],iMotor:=2);
GVL.pm[3].outConv.belt[1].fbconverter(stConverter:= GVL.stConverter[5],iMotor:=3);
GVL.pm[4].inConv.belt[0].fbconverter(stConverter:= GVL.stConverter[6],iMotor:=0);
GVL.pm[4].inConv.belt[1].fbconverter(stConverter:= GVL.stConverter[6],iMotor:=1);
GVL.pm[4].inConv.belt[2].fbconverter(stConverter:= GVL.stConverter[6],iMotor:=2);
GVL.pm[5].inConv.belt[0].fbconverter(stConverter:= GVL.stConverter[6],iMotor:=3);
GVL.pm[5].inConv.belt[1].fbconverter(stConverter:= GVL.stConverter[6],iMotor:=4);
GVL.pm[5].inConv.belt[2].fbconverter(stConverter:= GVL.stConverter[6],iMotor:=5);
GVL.pm[4].outConv.belt[0].fbconverter(stConverter:= GVL.stConverter[7],iMotor:=0);
GVL.pm[4].outConv.belt[1].fbconverter(stConverter:= GVL.stConverter[7],iMotor:=1);
GVL.pm[5].outConv.belt[0].fbconverter(stConverter:= GVL.stConverter[7],iMotor:=2);
GVL.pm[5].outConv.belt[1].fbconverter(stConverter:= GVL.stConverter[7],iMotor:=3);
GVL.pm[6].inConv.belt[0].fbconverter(stConverter:= GVL.stConverter[8],iMotor:=0);
GVL.pm[6].inConv.belt[1].fbconverter(stConverter:= GVL.stConverter[8],iMotor:=1);
GVL.pm[6].inConv.belt[2].fbconverter(stConverter:= GVL.stConverter[8],iMotor:=2);
GVL.pm[7].inConv.belt[0].fbconverter(stConverter:= GVL.stConverter[8],iMotor:=3);
GVL.pm[7].inConv.belt[1].fbconverter(stConverter:= GVL.stConverter[8],iMotor:=4);
GVL.pm[7].inConv.belt[2].fbconverter(stConverter:= GVL.stConverter[8],iMotor:=5);
GVL.pm[6].outConv.belt[0].fbconverter(stConverter:= GVL.stConverter[9],iMotor:=0);
GVL.pm[6].outConv.belt[1].fbconverter(stConverter:= GVL.stConverter[9],iMotor:=1);
GVL.pm[7].outConv.belt[0].fbconverter(stConverter:= GVL.stConverter[9],iMotor:=2);
GVL.pm[7].outConv.belt[1].fbconverter(stConverter:= GVL.stConverter[9],iMotor:=3);
GVL.pm[8].inConv.belt[0].fbconverter(stConverter:= GVL.stConverter[10],iMotor:=0);
GVL.pm[8].inConv.belt[1].fbconverter(stConverter:= GVL.stConverter[10],iMotor:=1);
GVL.pm[8].inConv.belt[2].fbconverter(stConverter:= GVL.stConverter[10],iMotor:=2);
GVL.pm[9].inConv.belt[0].fbconverter(stConverter:= GVL.stConverter[10],iMotor:=3);
GVL.pm[9].inConv.belt[1].fbconverter(stConverter:= GVL.stConverter[10],iMotor:=4);
GVL.pm[9].inConv.belt[2].fbconverter(stConverter:= GVL.stConverter[10],iMotor:=5);
GVL.pm[8].outConv.belt[0].fbconverter(stConverter:= GVL.stConverter[11],iMotor:=0);
GVL.pm[8].outConv.belt[1].fbconverter(stConverter:= GVL.stConverter[11],iMotor:=1);
GVL.pm[9].outConv.belt[0].fbconverter(stConverter:= GVL.stConverter[11],iMotor:=2);
GVL.pm[9].outConv.belt[1].fbconverter(stConverter:= GVL.stConverter[11],iMotor:=3);
GVL.lb[1].belt[0].fbconverter(stConverter:=GVL.stConverter[12],iMotor:=0);
GVL.lb[1].belt[1].fbconverter(stConverter:=GVL.stConverter[12],iMotor:=1);
GVL.lb[1].belt[2].fbconverter(stConverter:=GVL.stConverter[12],iMotor:=2);
GVL.lc[1].belt_out.belt.fbconverter(stConverter:=GVL.stConverter[13],iMotor:=0);



GVL.ref_fbconverterMotor[0]		:= ADR(GVL.lb[0].belt[0].fbconverter);
GVL.ref_fbconverterMotor[1]		:= ADR(GVL.lb[0].belt[1].fbconverter);
GVL.ref_fbconverterMotor[2]		:= ADR(GVL.lb[0].belt[2].fbconverter);
GVL.ref_fbconverterMotor[3]		:= ADR(GVL.lc[0].belt_out.belt.fbconverter);
GVL.ref_fbconverterMotor[4]		:= ADR(GVL.pm[0].inConv.belt[0].fbconverter);
GVL.ref_fbconverterMotor[5]		:= ADR(GVL.pm[0].inConv.belt[1].fbconverter);
GVL.ref_fbconverterMotor[6]		:= ADR(GVL.pm[0].inConv.belt[2].fbconverter);
GVL.ref_fbconverterMotor[7]		:= ADR(GVL.pm[1].inConv.belt[0].fbconverter);
GVL.ref_fbconverterMotor[8]		:= ADR(GVL.pm[1].inConv.belt[1].fbconverter);
GVL.ref_fbconverterMotor[9]		:= ADR(GVL.pm[1].inConv.belt[2].fbconverter);
GVL.ref_fbconverterMotor[10]	:= ADR(GVL.pm[0].outConv.belt[0].fbconverter);
GVL.ref_fbconverterMotor[11]	:= ADR(GVL.pm[0].outConv.belt[1].fbconverter);
GVL.ref_fbconverterMotor[12]	:= ADR(GVL.pm[1].outConv.belt[0].fbconverter);
GVL.ref_fbconverterMotor[13]	:= ADR(GVL.pm[1].outConv.belt[1].fbconverter);
GVL.ref_fbconverterMotor[14]	:= ADR(GVL.pm[2].inConv.belt[0].fbconverter);
GVL.ref_fbconverterMotor[15]	:= ADR(GVL.pm[2].inConv.belt[1].fbconverter);
GVL.ref_fbconverterMotor[16]	:= ADR(GVL.pm[2].inConv.belt[2].fbconverter);
GVL.ref_fbconverterMotor[17]	:= ADR(GVL.pm[3].inConv.belt[0].fbconverter);
GVL.ref_fbconverterMotor[18]	:= ADR(GVL.pm[3].inConv.belt[1].fbconverter);
GVL.ref_fbconverterMotor[19]	:= ADR(GVL.pm[3].inConv.belt[2].fbconverter);
GVL.ref_fbconverterMotor[20]	:= ADR(GVL.pm[2].outConv.belt[0].fbconverter);
GVL.ref_fbconverterMotor[21]	:= ADR(GVL.pm[2].outConv.belt[1].fbconverter);
GVL.ref_fbconverterMotor[22]	:= ADR(GVL.pm[3].outConv.belt[0].fbconverter);
GVL.ref_fbconverterMotor[23]	:= ADR(GVL.pm[3].outConv.belt[1].fbconverter);
GVL.ref_fbconverterMotor[24]	:= ADR(GVL.pm[4].inConv.belt[0].fbconverter);
GVL.ref_fbconverterMotor[25]	:= ADR(GVL.pm[4].inConv.belt[1].fbconverter);
GVL.ref_fbconverterMotor[26]	:= ADR(GVL.pm[4].inConv.belt[2].fbconverter);
GVL.ref_fbconverterMotor[27]	:= ADR(GVL.pm[5].inConv.belt[0].fbconverter);
GVL.ref_fbconverterMotor[28]	:= ADR(GVL.pm[5].inConv.belt[1].fbconverter);
GVL.ref_fbconverterMotor[29]	:= ADR(GVL.pm[5].inConv.belt[2].fbconverter);
GVL.ref_fbconverterMotor[30]	:= ADR(GVL.pm[4].outConv.belt[0].fbconverter);
GVL.ref_fbconverterMotor[31]	:= ADR(GVL.pm[4].outConv.belt[1].fbconverter);
GVL.ref_fbconverterMotor[32]	:= ADR(GVL.pm[5].outConv.belt[0].fbconverter);
GVL.ref_fbconverterMotor[33]	:= ADR(GVL.pm[5].outConv.belt[1].fbconverter);
GVL.ref_fbconverterMotor[34]	:= ADR(GVL.pm[6].inConv.belt[0].fbconverter);
GVL.ref_fbconverterMotor[35]	:= ADR(GVL.pm[6].inConv.belt[1].fbconverter);
GVL.ref_fbconverterMotor[36]	:= ADR(GVL.pm[6].inConv.belt[2].fbconverter);
GVL.ref_fbconverterMotor[37]	:= ADR(GVL.pm[7].inConv.belt[0].fbconverter);
GVL.ref_fbconverterMotor[38]	:= ADR(GVL.pm[7].inConv.belt[1].fbconverter);
GVL.ref_fbconverterMotor[39]	:= ADR(GVL.pm[7].inConv.belt[2].fbconverter);
GVL.ref_fbconverterMotor[40]	:= ADR(GVL.pm[6].outConv.belt[0].fbconverter);
GVL.ref_fbconverterMotor[41]	:= ADR(GVL.pm[6].outConv.belt[1].fbconverter);
GVL.ref_fbconverterMotor[42]	:= ADR(GVL.pm[7].outConv.belt[0].fbconverter);
GVL.ref_fbconverterMotor[43]	:= ADR(GVL.pm[7].outConv.belt[1].fbconverter);
GVL.ref_fbconverterMotor[44]	:= ADR(GVL.pm[8].inConv.belt[0].fbconverter);
GVL.ref_fbconverterMotor[45]	:= ADR(GVL.pm[8].inConv.belt[1].fbconverter);
GVL.ref_fbconverterMotor[46]	:= ADR(GVL.pm[8].inConv.belt[2].fbconverter);
GVL.ref_fbconverterMotor[47]	:= ADR(GVL.pm[9].inConv.belt[0].fbconverter);
GVL.ref_fbconverterMotor[48]	:= ADR(GVL.pm[9].inConv.belt[1].fbconverter);
GVL.ref_fbconverterMotor[49]	:= ADR(GVL.pm[9].inConv.belt[2].fbconverter);
GVL.ref_fbconverterMotor[50]	:= ADR(GVL.pm[8].outConv.belt[0].fbconverter);
GVL.ref_fbconverterMotor[51]	:= ADR(GVL.pm[8].outConv.belt[1].fbconverter);
GVL.ref_fbconverterMotor[52]	:= ADR(GVL.pm[9].outConv.belt[0].fbconverter);
GVL.ref_fbconverterMotor[53]	:= ADR(GVL.pm[9].outConv.belt[1].fbconverter);
GVL.ref_fbconverterMotor[54]	:= ADR(GVL.lb[1].belt[0].fbconverter);
GVL.ref_fbconverterMotor[55]	:= ADR(GVL.lb[1].belt[1].fbconverter);
GVL.ref_fbconverterMotor[56]	:= ADR(GVL.lb[1].belt[2].fbconverter);
GVL.ref_fbconverterMotor[57]	:= ADR(GVL.lc[1].belt_out.belt.fbconverter);


